LIN {X 0,Y 330.91,Z 992.639,A -85,B 0,C 180,E1 15009.118,E2 15009.118} C_VEL
LIN {X 0,Y 333.093,Z 983.84,A -85,B 0,C 180,E1 15005.534,E2 15005.534} C_VEL
LIN {X 0,Y 336.451,Z 972.211,A -85,B 0,C 180,E1 15001.598,E2 15001.598} C_VEL
LIN {X 0,Y 340.194,Z 960.433,A -85,B 0,C 180,E1 14998.264,E2 14998.264} C_VEL
LIN {X 0,Y 344.804,Z 946.621,A -85,B 0,C 180,E1 14994.966,E2 14994.966} C_VEL
LIN {X 0,Y 350.006,Z 931.551,A -85,B 0,C 180,E1 14991.906,E2 14991.906} C_VEL
LIN {X 0,Y 355.638,Z 914.95,A -85,B 0,C 180,E1 14989.083,E2 14989.083} C_VEL
LIN {X 0,Y 361.606,Z 897.07,A -85,B 0,C 180,E1 14986.496,E2 14986.496} C_VEL
LIN {X 0,Y 367.141,Z 879.555,A -85,B 0,C 180,E1 14984.374,E2 14984.374} C_VEL
LIN {X 0,Y 373.38,Z 858.51,A -85,B 0,C 180,E1 14982.232,E2 14982.232} C_VEL
LIN {X 0,Y 378.589,Z 839.318,A -85,B 0,C 180,E1 14980.607,E2 14980.607} C_VEL
LIN {X 0,Y 383.892,Z 817.228,A -85,B 0,C 180,E1 14979.071,E2 14979.071} C_VEL
LIN {X 0,Y 388.44,Z 795.784,A -85,B 0,C 180,E1 14977.862,E2 14977.862} C_VEL
LIN {X 0,Y 392.348,Z 773.028,A -85,B 0,C 180,E1 14976.87,E2 14976.87} C_VEL
LIN {X 0,Y 395.641,Z 749.252,A -85,B 0,C 180,E1 14976.094,E2 14976.094} C_VEL
LIN {X 0,Y 397.692,Z 726.736,A -85,B 0,C 180,E1 14975.556,E2 14975.556} C_VEL
LIN {X 0,Y 410.028,Z 517.167,A -85,B 0,C 180,E1 14971.398,E2 14971.398} C_VEL
LIN {X 0,Y 411.387,Z 493.975,A -85,B 0,C 180,E1 14970.919,E2 14970.919} C_VEL
LIN {X 0,Y 401.273,Z 477.851,A -85,B 0,C 180,E1 14968.094,E2 14968.094} C_VEL
LIN {X 0,Y 391.227,Z 463.001,A -85,B 0,C 180,E1 14964.981,E2 14964.981} C_VEL
LIN {X 0,Y 382.41,Z 450.658,A -85,B 0,C 180,E1 14961.915,E2 14961.915} C_VEL
LIN {X 0,Y 378.241,Z 445.412,A -85,B 0,C 180,E1 14960.341,E2 14960.341} C_VEL
LIN {X 0,Y 374.323,Z 440.519,A -85,B 0,C 180,E1 14958.775,E2 14958.775} C_VEL
LIN {X 0,Y 370.45,Z 435.602,A -85,B 0,C 180,E1 14957.109,E2 14957.109} C_VEL
LIN {X 0,Y 366.394,Z 431.101,A -85,B 0,C 180,E1 14955.268,E2 14955.268} C_VEL
LIN {X 0,Y 364.882,Z 429.094,A -85,B 0,C 180,E1 14954.52,E2 14954.52} C_VEL
LIN {X 0,Y 361.373,Z 425.41,A -85,B 0,C 180,E1 14952.747,E2 14952.747} C_VEL
LIN {X 0,Y 359.797,Z 423.107,A -85,B 0,C 180,E1 14951.867,E2 14951.867} C_VEL
LIN {X 0,Y 356.404,Z 419.891,A -85,B 0,C 180,E1 14949.935,E2 14949.935} C_VEL
LIN {X 0,Y 354.609,Z 416.906,A -85,B 0,C 180,E1 14948.757,E2 14948.757} C_VEL
LIN {X 0,Y 351.319,Z 414.41,A -85,B 0,C 180,E1 14946.618,E2 14946.618} C_VEL
LIN {X 0,Y 349.107,Z 410.908,A -85,B 0,C 180,E1 14944.887,E2 14944.887} C_VEL
LIN {X 0,Y 348.552,Z 410.26,A -85,B 0,C 180,E1 14944.442,E2 14944.442} C_VEL
LIN {X 0,Y 345.174,Z 407.913,A -85,B 0,C 180,E1 14941.659,E2 14941.659} C_VEL
LIN {X 0,Y 342.781,Z 403.846,A -85,B 0,C 180,E1 14938.997,E2 14938.997} C_VEL
LIN {X 0,Y 338.729,Z 401.153,A -85,B 0,C 180,E1 14933.729,E2 14933.729} C_VEL
LIN {X 0,Y 336.722,Z 397.551,A -85,B 0,C 180,E1 14928.46,E2 14928.46} C_VEL
LIN {X 0,Y 336.018,Z 396.934,A -85,B 0,C 180,E1 14923.757,E2 14923.757} C_VEL
LIN {X 0,Y 336.593,Z 397.417,A -85,B 0,C 180,E1 14919.116,E2 14919.116} C_VEL
LIN {X 0,Y 337.44,Z 399.091,A -85,B 0,C 180,E1 14916.235,E2 14916.235} C_VEL
LIN {X 0,Y 340.379,Z 402.576,A -85,B 0,C 180,E1 14911.008,E2 14911.008} C_VEL
LIN {X 0,Y 343.088,Z 404.15,A -85,B 0,C 180,E1 14907.868,E2 14907.868} C_VEL
LIN {X 0,Y 345.313,Z 408.031,A -85,B 0,C 180,E1 14905.422,E2 14905.422} C_VEL
LIN {X 0,Y 349.089,Z 410.785,A -85,B 0,C 180,E1 14902.353,E2 14902.353} C_VEL
LIN {X 0,Y 351.324,Z 414.39,A -85,B 0,C 180,E1 14900.605,E2 14900.605} C_VEL
LIN {X 0,Y 354.877,Z 417.344,A -85,B 0,C 180,E1 14898.291,E2 14898.291} C_VEL
LIN {X 0,Y 357.657,Z 421.353,A -85,B 0,C 180,E1 14896.55,E2 14896.55} C_VEL
LIN {X 0,Y 360.381,Z 423.715,A -85,B 0,C 180,E1 14895.07,E2 14895.07} C_VEL
LIN {X 0,Y 363.451,Z 427.853,A -85,B 0,C 180,E1 14893.425,E2 14893.425} C_VEL
LIN {X 0,Y 365.762,Z 430.068,A -85,B 0,C 180,E1 14892.315,E2 14892.315} C_VEL
LIN {X 0,Y 369.415,Z 434.618,A -85,B 0,C 180,E1 14890.606,E2 14890.606} C_VEL
LIN {X 0,Y 371.075,Z 436.552,A -85,B 0,C 180,E1 14889.881,E2 14889.881} C_VEL
LIN {X 0,Y 375.981,Z 442.563,A -85,B 0,C 180,E1 14887.83,E2 14887.83} C_VEL
LIN {X 0,Y 380.704,Z 448.431,A -85,B 0,C 180,E1 14886.009,E2 14886.009} C_VEL
LIN {X 0,Y 385.386,Z 454.312,A -85,B 0,C 180,E1 14884.335,E2 14884.335} C_VEL
LIN {X 0,Y 393.083,Z 464.398,A -85,B 0,C 180,E1 14881.786,E2 14881.786} C_VEL
LIN {X 0,Y 402.393,Z 477.147,A -85,B 0,C 180,E1 14878.996,E2 14878.996} C_VEL
LIN {X 0,Y 411.104,Z 489.93,A -85,B 0,C 180,E1 14876.615,E2 14876.615} C_VEL
LIN {X 0,Y 398.81,Z 697.255,A -85,B 0,C 180,E1 14872.515,E2 14872.515} C_VEL
LIN {X 0,Y 396.721,Z 724.489,A -85,B 0,C 180,E1 14871.906,E2 14871.906} C_VEL
LIN {X 0,Y 393.982,Z 747.489,A -85,B 0,C 180,E1 14871.191,E2 14871.191} C_VEL
LIN {X 0,Y 390.444,Z 769.449,A -85,B 0,C 180,E1 14870.259,E2 14870.259} C_VEL
LIN {X 0,Y 386.299,Z 791.019,A -85,B 0,C 180,E1 14869.107,E2 14869.107} C_VEL
LIN {X 0,Y 381.676,Z 811.199,A -85,B 0,C 180,E1 14867.765,E2 14867.765} C_VEL
LIN {X 0,Y 376.156,Z 832.56,A -85,B 0,C 180,E1 14866.043,E2 14866.043} C_VEL
LIN {X 0,Y 370.908,Z 850.781,A -85,B 0,C 180,E1 14864.275,E2 14864.275} C_VEL
LIN {X 0,Y 364.791,Z 870.313,A -85,B 0,C 180,E1 14862.019,E2 14862.019} C_VEL
LIN {X 0,Y 359.17,Z 887.26,A -85,B 0,C 180,E1 14859.691,E2 14859.691} C_VEL
LIN {X 0,Y 355.793,Z 896.961,A -85,B 0,C 180,E1 14858.165,E2 14858.165} C_VEL
LIN {X 0,Y 353.148,Z 902.367,A -85,B 0,C 180,E1 14857.37,E2 14857.37} C_VEL
LIN {X 0,Y 343.413,Z 915.776,A -85,B 0,C 180,E1 14855.488,E2 14855.488} C_VEL
LIN {X 0,Y 340.743,Z 920.57,A -85,B 0,C 180,E1 14854.568,E2 14854.568} C_VEL
LIN {X 0,Y 335.906,Z 933.491,A -85,B 0,C 180,E1 14851.531,E2 14851.531} C_VEL
LIN {X 0,Y 330.984,Z 947.025,A -85,B 0,C 180,E1 14847.745,E2 14847.745} C_VEL
LIN {X 0,Y 327.238,Z 958.049,A -85,B 0,C 180,E1 14844.033,E2 14844.033} C_VEL
LIN {X 0,Y 324.369,Z 967.228,A -85,B 0,C 180,E1 14840.235,E2 14840.235} C_VEL
LIN {X 0,Y 322.352,Z 974.985,A -85,B 0,C 180,E1 14836.361,E2 14836.361} C_VEL
LIN {X 0,Y 321.026,Z 981.137,A -85,B 0,C 180,E1 14832.376,E2 14832.376} C_VEL
LIN {X 0,Y 320.326,Z 985.864,A -85,B 0,C 180,E1 14828.384,E2 14828.384} C_VEL
LIN {X 0,Y 320.045,Z 988.794,A -85,B 0,C 180,E1 14824.655,E2 14824.655} C_VEL
LIN {X 0,Y 319.986,Z 990.509,A -85,B 0,C 180,E1 14821.027,E2 14821.027} C_VEL
LIN {X 0,Y 319.956,Z 990.924,A -85,B 0,C 180,E1 14817.057,E2 14817.057} C_VEL
LIN {X 0,Y 319.974,Z 990.17,A -85,B 0,C 180,E1 14813.727,E2 14813.727} C_VEL
LIN {X 0,Y 320.14,Z 988.143,A -85,B 0,C 180,E1 14809.924,E2 14809.924} C_VEL
LIN {X 0,Y 320.531,Z 984.612,A -85,B 0,C 180,E1 14806.103,E2 14806.103} C_VEL
LIN {X 0,Y 321.437,Z 979.74,A -85,B 0,C 180,E1 14802.214,E2 14802.214} C_VEL
LIN {X 0,Y 322.994,Z 973.105,A -85,B 0,C 180,E1 14798.253,E2 14798.253} C_VEL
LIN {X 0,Y 325.442,Z 964.846,A -85,B 0,C 180,E1 14794.259,E2 14794.259} C_VEL
LIN {X 0,Y 328.74,Z 954.945,A -85,B 0,C 180,E1 14790.426,E2 14790.426} C_VEL
LIN {X 0,Y 333.353,Z 942.442,A -85,B 0,C 180,E1 14786.423,E2 14786.423} C_VEL
LIN {X 0,Y 338.143,Z 930.095,A -85,B 0,C 180,E1 14783.126,E2 14783.126} C_VEL
LIN {X 0,Y 343.659,Z 916.024,A -85,B 0,C 180,E1 14779.983,E2 14779.983} C_VEL
LIN {X 0,Y 349.738,Z 900.54,A -85,B 0,C 180,E1 14777.04,E2 14777.04} C_VEL
LIN {X 0,Y 355.801,Z 884.413,A -85,B 0,C 180,E1 14774.484,E2 14774.484} C_VEL
LIN {X 0,Y 362.443,Z 866.085,A -85,B 0,C 180,E1 14772.022,E2 14772.022} C_VEL
LIN {X 0,Y 368.203,Z 848.908,A -85,B 0,C 180,E1 14770.088,E2 14770.088} C_VEL
LIN {X 0,Y 374.697,Z 827.854,A -85,B 0,C 180,E1 14768.099,E2 14768.099} C_VEL
LIN {X 0,Y 380.15,Z 808.098,A -85,B 0,C 180,E1 14766.563,E2 14766.563} C_VEL
LIN {X 0,Y 385.245,Z 786.857,A -85,B 0,C 180,E1 14765.212,E2 14765.212} C_VEL
LIN {X 0,Y 389.81,Z 764.653,A -85,B 0,C 180,E1 14764.078,E2 14764.078} C_VEL
LIN {X 0,Y 393.502,Z 741.577,A -85,B 0,C 180,E1 14763.184,E2 14763.184} C_VEL
LIN {X 0,Y 396.477,Z 716.689,A -85,B 0,C 180,E1 14762.486,E2 14762.486} C_VEL
LIN {X 0,Y 412.263,Z 510.138,A -85,B 0,C 180,E1 14758.198,E2 14758.198} C_VEL
LIN {X 0,Y 413.31,Z 496.471,A -85,B 0,C 180,E1 14757.89,E2 14757.89} C_VEL
LIN {X 0,Y 407.813,Z 487.013,A -85,B 0,C 180,E1 14755.501,E2 14755.501} C_VEL
LIN {X 0,Y 403.867,Z 480.436,A -85,B 0,C 180,E1 14753.39,E2 14753.39} C_VEL
LIN {X 0,Y 401.279,Z 476.234,A -85,B 0,C 180,E1 14751.691,E2 14751.691} C_VEL
LIN {X 0,Y 398.884,Z 472.1,A -85,B 0,C 180,E1 14749.603,E2 14749.603} C_VEL
LIN {X 0,Y 396.705,Z 468.572,A -85,B 0,C 180,E1 14746.444,E2 14746.444} C_VEL
LIN {X 0,Y 396.482,Z 467.384,A -85,B 0,C 180,E1 14745.394,E2 14745.394} C_VEL
LIN {X 0,Y 396.528,Z 467.443,A -85,B 0,C 180,E1 14742.842,E2 14742.842} C_VEL
LIN {X 0,Y 398.037,Z 471.243,A -85,B 0,C 180,E1 14739.718,E2 14739.718} C_VEL
LIN {X 0,Y 399.24,Z 472.726,A -85,B 0,C 180,E1 14738.476,E2 14738.476} C_VEL
LIN {X 0,Y 402.217,Z 477.734,A -85,B 0,C 180,E1 14736.097,E2 14736.097} C_VEL
LIN {X 0,Y 405.36,Z 483.575,A -85,B 0,C 180,E1 14734.157,E2 14734.157} C_VEL
LIN {X 0,Y 409.464,Z 491.64,A -85,B 0,C 180,E1 14732.085,E2 14732.085} C_VEL
LIN {X 0,Y 413.288,Z 499.593,A -85,B 0,C 180,E1 14730.423,E2 14730.423} C_VEL
LIN {X 0,Y 399.434,Z 680.245,A -85,B 0,C 180,E1 14726.677,E2 14726.677} C_VEL
LIN {X 0,Y 395.3,Z 735.513,A -85,B 0,C 180,E1 14725.506,E2 14725.506} C_VEL
LIN {X 0,Y 392.181,Z 758.741,A -85,B 0,C 180,E1 14724.843,E2 14724.843} C_VEL
LIN {X 0,Y 388.044,Z 782.281,A -85,B 0,C 180,E1 14723.946,E2 14723.946} C_VEL
LIN {X 0,Y 383.894,Z 801.848,A -85,B 0,C 180,E1 14722.983,E2 14722.983} C_VEL
LIN {X 0,Y 378.352,Z 824.459,A -85,B 0,C 180,E1 14721.591,E2 14721.591} C_VEL
LIN {X 0,Y 373.178,Z 843.178,A -85,B 0,C 180,E1 14720.182,E2 14720.182} C_VEL
LIN {X 0,Y 366.642,Z 864.591,A -85,B 0,C 180,E1 14718.236,E2 14718.236} C_VEL
LIN {X 0,Y 360.423,Z 883.572,A -85,B 0,C 180,E1 14716.164,E2 14716.164} C_VEL
LIN {X 0,Y 354.049,Z 901.749,A -85,B 0,C 180,E1 14713.784,E2 14713.784} C_VEL
LIN {X 0,Y 347.941,Z 918.842,A -85,B 0,C 180,E1 14711.156,E2 14711.156} C_VEL
LIN {X 0,Y 341.813,Z 935.354,A -85,B 0,C 180,E1 14708.117,E2 14708.117} C_VEL
LIN {X 0,Y 336.304,Z 950.548,A -85,B 0,C 180,E1 14704.812,E2 14704.812} C_VEL
LIN {X 0,Y 331.687,Z 963.637,A -85,B 0,C 180,E1 14701.437,E2 14701.437} C_VEL
LIN {X 0,Y 327.626,Z 975.984,A -85,B 0,C 180,E1 14697.642,E2 14697.642} C_VEL
LIN {X 0,Y 324.704,Z 985.988,A -85,B 0,C 180,E1 14693.987,E2 14693.987} C_VEL
LIN {X 0,Y 322.437,Z 995.015,A -85,B 0,C 180,E1 14689.948,E2 14689.948} C_VEL
LIN {X 0,Y 321.025,Z 1002.362,A -85,B 0,C 180,E1 14685.912,E2 14685.912} C_VEL
LIN {X 0,Y 320.293,Z 1007.625,A -85,B 0,C 180,E1 14682.077,E2 14682.077} C_VEL
LIN {X 0,Y 320.032,Z 1011.372,A -85,B 0,C 180,E1 14678.448,E2 14678.448} C_VEL
LIN {X 0,Y 319.948,Z 1013.912,A -85,B 0,C 180,E1 14674.485,E2 14674.485} C_VEL
LIN {X 0,Y 319.955,Z 1014.848,A -85,B 0,C 180,E1 14671.258,E2 14671.258} C_VEL
LIN {X 0,Y 319.957,Z 1014.757,A -85,B 0,C 180,E1 14667.856,E2 14667.856} C_VEL
LIN {X 0,Y 319.959,Z 1013.149,A -85,B 0,C 180,E1 14663.906,E2 14663.906} C_VEL
LIN {X 0,Y 320.069,Z 1010.511,A -85,B 0,C 180,E1 14660.475,E2 14660.475} C_VEL
LIN {X 0,Y 320.522,Z 1006.032,A -85,B 0,C 180,E1 14656.475,E2 14656.475} C_VEL
LIN {X 0,Y 321.456,Z 1000.106,A -85,B 0,C 180,E1 14652.632,E2 14652.632} C_VEL
LIN {X 0,Y 323.158,Z 992.282,A -85,B 0,C 180,E1 14648.592,E2 14648.592} C_VEL
LIN {X 0,Y 325.502,Z 983.467,A -85,B 0,C 180,E1 14644.925,E2 14644.925} C_VEL
LIN {X 0,Y 329.077,Z 971.865,A -85,B 0,C 180,E1 14640.919,E2 14640.919} C_VEL
LIN {X 0,Y 333.072,Z 960.003,A -85,B 0,C 180,E1 14637.504,E2 14637.504} C_VEL
LIN {X 0,Y 337.94,Z 946.141,A -85,B 0,C 180,E1 14634.146,E2 14634.146} C_VEL
LIN {X 0,Y 343.504,Z 930.845,A -85,B 0,C 180,E1 14631.002,E2 14631.002} C_VEL
LIN {X 0,Y 349.325,Z 914.383,A -85,B 0,C 180,E1 14628.179,E2 14628.179} C_VEL
LIN {X 0,Y 355.575,Z 896.402,A -85,B 0,C 180,E1 14625.567,E2 14625.567} C_VEL
LIN {X 0,Y 361.579,Z 878.166,A -85,B 0,C 180,E1 14623.351,E2 14623.351} C_VEL
LIN {X 0,Y 367.893,Z 857.519,A -85,B 0,C 180,E1 14621.254,E2 14621.254} C_VEL
LIN {X 0,Y 373.243,Z 838.445,A -85,B 0,C 180,E1 14619.64,E2 14619.64} C_VEL
LIN {X 0,Y 378.399,Z 817.624,A -85,B 0,C 180,E1 14618.192,E2 14618.192} C_VEL
LIN {X 0,Y 383.162,Z 795.876,A -85,B 0,C 180,E1 14616.96,E2 14616.96} C_VEL
LIN {X 0,Y 387.235,Z 772.987,A -85,B 0,C 180,E1 14615.957,E2 14615.957} C_VEL
LIN {X 0,Y 390.634,Z 749.321,A -85,B 0,C 180,E1 14615.182,E2 14615.182} C_VEL
LIN {X 0,Y 392.766,Z 726.741,A -85,B 0,C 180,E1 14614.638,E2 14614.638} C_VEL
LIN {X 0,Y 405.62,Z 516.743,A -85,B 0,C 180,E1 14610.449,E2 14610.449} C_VEL
LIN {X 0,Y 406.726,Z 498.175,A -85,B 0,C 180,E1 14610.062,E2 14610.062} C_VEL
LIN {X 0,Y 397.976,Z 484.066,A -85,B 0,C 180,E1 14607.533,E2 14607.533} C_VEL
LIN {X 0,Y 388.403,Z 469.686,A -85,B 0,C 180,E1 14604.485,E2 14604.485} C_VEL
LIN {X 0,Y 379.904,Z 457.646,A -85,B 0,C 180,E1 14601.458,E2 14601.458} C_VEL
LIN {X 0,Y 375.865,Z 452.522,A -85,B 0,C 180,E1 14599.907,E2 14599.907} C_VEL
LIN {X 0,Y 372.014,Z 447.669,A -85,B 0,C 180,E1 14598.328,E2 14598.328} C_VEL
LIN {X 0,Y 367.517,Z 442.164,A -85,B 0,C 180,E1 14596.354,E2 14596.354} C_VEL
LIN {X 0,Y 363.777,Z 437.473,A -85,B 0,C 180,E1 14594.565,E2 14594.565} C_VEL
LIN {X 0,Y 359.268,Z 432.497,A -85,B 0,C 180,E1 14592.251,E2 14592.251} C_VEL
LIN {X 0,Y 358.132,Z 430.776,A -85,B 0,C 180,E1 14591.596,E2 14591.596} C_VEL
LIN {X 0,Y 354.635,Z 427.367,A -85,B 0,C 180,E1 14589.575,E2 14589.575} C_VEL
LIN {X 0,Y 352.73,Z 424.487,A -85,B 0,C 180,E1 14588.312,E2 14588.312} C_VEL
LIN {X 0,Y 349.419,Z 421.648,A -85,B 0,C 180,E1 14586.077,E2 14586.077} C_VEL
LIN {X 0,Y 347.235,Z 418.11,A -85,B 0,C 180,E1 14584.293,E2 14584.293} C_VEL
LIN {X 0,Y 343.702,Z 415.553,A -85,B 0,C 180,E1 14581.333,E2 14581.333} C_VEL
LIN {X 0,Y 341.496,Z 411.677,A -85,B 0,C 180,E1 14578.825,E2 14578.825} C_VEL
LIN {X 0,Y 337.513,Z 408.987,A -85,B 0,C 180,E1 14573.536,E2 14573.536} C_VEL
LIN {X 0,Y 335.565,Z 405.439,A -85,B 0,C 180,E1 14568.31,E2 14568.31} C_VEL
LIN {X 0,Y 334.91,Z 404.851,A -85,B 0,C 180,E1 14563.523,E2 14563.523} C_VEL
LIN {X 0,Y 335.611,Z 405.454,A -85,B 0,C 180,E1 14558.686,E2 14558.686} C_VEL
LIN {X 0,Y 338.405,Z 409.854,A -85,B 0,C 180,E1 14552.171,E2 14552.171} C_VEL
LIN {X 0,Y 341.724,Z 411.891,A -85,B 0,C 180,E1 14548.12,E2 14548.12} C_VEL
LIN {X 0,Y 343.957,Z 415.81,A -85,B 0,C 180,E1 14545.635,E2 14545.635} C_VEL
LIN {X 0,Y 347.537,Z 418.459,A -85,B 0,C 180,E1 14542.675,E2 14542.675} C_VEL
LIN {X 0,Y 350.003,Z 422.307,A -85,B 0,C 180,E1 14540.72,E2 14540.72} C_VEL
LIN {X 0,Y 353.228,Z 425.038,A -85,B 0,C 180,E1 14538.592,E2 14538.592} C_VEL
LIN {X 0,Y 356.131,Z 429.107,A -85,B 0,C 180,E1 14536.76,E2 14536.76} C_VEL
LIN {X 0,Y 358.645,Z 431.399,A -85,B 0,C 180,E1 14535.368,E2 14535.368} C_VEL
LIN {X 0,Y 361.874,Z 435.618,A -85,B 0,C 180,E1 14533.621,E2 14533.621} C_VEL
LIN {X 0,Y 363.902,Z 437.65,A -85,B 0,C 180,E1 14532.635,E2 14532.635} C_VEL
LIN {X 0,Y 367.605,Z 442.217,A -85,B 0,C 180,E1 14530.874,E2 14530.874} C_VEL
LIN {X 0,Y 373.794,Z 449.865,A -85,B 0,C 180,E1 14528.209,E2 14528.209} C_VEL
LIN {X 0,Y 378.705,Z 456.06,A -85,B 0,C 180,E1 14526.286,E2 14526.286} C_VEL
LIN {X 0,Y 383.771,Z 462.499,A -85,B 0,C 180,E1 14524.452,E2 14524.452} C_VEL
LIN {X 0,Y 393.127,Z 474.956,A -85,B 0,C 180,E1 14521.358,E2 14521.358} C_VEL
LIN {X 0,Y 403.739,Z 490.155,A -85,B 0,C 180,E1 14518.225,E2 14518.225} C_VEL
LIN {X 0,Y 406.441,Z 494.536,A -85,B 0,C 180,E1 14517.468,E2 14517.468} C_VEL
LIN {X 0,Y 393.64,Z 702.589,A -85,B 0,C 180,E1 14513.331,E2 14513.331} C_VEL
LIN {X 0,Y 391.59,Z 726.521,A -85,B 0,C 180,E1 14512.772,E2 14512.772} C_VEL
LIN {X 0,Y 388.641,Z 749.694,A -85,B 0,C 180,E1 14512.027,E2 14512.027} C_VEL
LIN {X 0,Y 385.198,Z 770.255,A -85,B 0,C 180,E1 14511.144,E2 14511.144} C_VEL
LIN {X 0,Y 380.794,Z 792.284,A -85,B 0,C 180,E1 14509.954,E2 14509.954} C_VEL
LIN {X 0,Y 376.03,Z 812.406,A -85,B 0,C 180,E1 14508.602,E2 14508.602} C_VEL
LIN {X 0,Y 370.317,Z 833.635,A -85,B 0,C 180,E1 14506.868,E2 14506.868} C_VEL
LIN {X 0,Y 364.887,Z 851.797,A -85,B 0,C 180,E1 14505.084,E2 14505.084} C_VEL
LIN {X 0,Y 358.535,Z 871.225,A -85,B 0,C 180,E1 14502.804,E2 14502.804} C_VEL
LIN {X 0,Y 352.523,Z 888.687,A -85,B 0,C 180,E1 14500.371,E2 14500.371} C_VEL
LIN {X 0,Y 346.505,Z 905.102,A -85,B 0,C 180,E1 14497.623,E2 14497.623} C_VEL
LIN {X 0,Y 340.743,Z 920.57,A -85,B 0,C 180,E1 14494.568,E2 14494.568} C_VEL
LIN {X 0,Y 338.108,Z 925.306,A -85,B 0,C 180,E1 14493.617,E2 14493.617} C_VEL
LIN {X 0,Y 328.091,Z 937.671,A -85,B 0,C 180,E1 14491.193,E2 14491.193} C_VEL
LIN {X 0,Y 326.075,Z 941.156,A -85,B 0,C 180,E1 14490.277,E2 14490.277} C_VEL
LIN {X 0,Y 321.565,Z 953.258,A -85,B 0,C 180,E1 14486.478,E2 14486.478} C_VEL
LIN {X 0,Y 318.181,Z 962.982,A -85,B 0,C 180,E1 14482.775,E2 14482.775} C_VEL
LIN {X 0,Y 315.454,Z 971.82,A -85,B 0,C 180,E1 14478.662,E2 14478.662} C_VEL
LIN {X 0,Y 313.768,Z 978.407,A -85,B 0,C 180,E1 14474.848,E2 14474.848} C_VEL
LIN {X 0,Y 312.666,Z 984.079,A -85,B 0,C 180,E1 14470.57,E2 14470.57} C_VEL
LIN {X 0,Y 312.184,Z 987.545,A -85,B 0,C 180,E1 14466.995,E2 14466.995} C_VEL
LIN {X 0,Y 311.992,Z 990.13,A -85,B 0,C 180,E1 14462.926,E2 14462.926} C_VEL
LIN {X 0,Y 311.962,Z 991.137,A -85,B 0,C 180,E1 14459.358,E2 14459.358} C_VEL
LIN {X 0,Y 311.954,Z 991.102,A -85,B 0,C 180,E1 14455.877,E2 14455.877} C_VEL
LIN {X 0,Y 312.03,Z 989.685,A -85,B 0,C 180,E1 14451.793,E2 14451.793} C_VEL
LIN {X 0,Y 312.28,Z 987.245,A -85,B 0,C 180,E1 14448.238,E2 14448.238} C_VEL
LIN {X 0,Y 312.926,Z 983.148,A -85,B 0,C 180,E1 14444.152,E2 14444.152} C_VEL
LIN {X 0,Y 314.157,Z 977.592,A -85,B 0,C 180,E1 14440.191,E2 14440.191} C_VEL
LIN {X 0,Y 316.149,Z 970.673,A -85,B 0,C 180,E1 14436.243,E2 14436.243} C_VEL
LIN {X 0,Y 319.124,Z 961.659,A -85,B 0,C 180,E1 14432.184,E2 14432.184} C_VEL
LIN {X 0,Y 323.341,Z 950.407,A -85,B 0,C 180,E1 14428.037,E2 14428.037} C_VEL
LIN {X 0,Y 328.198,Z 938.354,A -85,B 0,C 180,E1 14424.363,E2 14424.363} C_VEL
LIN {X 0,Y 333.708,Z 924.882,A -85,B 0,C 180,E1 14420.97,E2 14420.97} C_VEL
LIN {X 0,Y 339.902,Z 910.055,A -85,B 0,C 180,E1 14417.815,E2 14417.815} C_VEL
LIN {X 0,Y 346.137,Z 894.608,A -85,B 0,C 180,E1 14415.069,E2 14415.069} C_VEL
LIN {X 0,Y 353.157,Z 876.566,A -85,B 0,C 180,E1 14412.365,E2 14412.365} C_VEL
LIN {X 0,Y 359.885,Z 858.283,A -85,B 0,C 180,E1 14410.081,E2 14410.081} C_VEL
LIN {X 0,Y 366.401,Z 838.867,A -85,B 0,C 180,E1 14408.071,E2 14408.071} C_VEL
LIN {X 0,Y 372.65,Z 818.56,A -85,B 0,C 180,E1 14406.316,E2 14406.316} C_VEL
LIN {X 0,Y 377.881,Z 798.972,A -85,B 0,C 180,E1 14404.934,E2 14404.934} C_VEL
LIN {X 0,Y 382.988,Z 777.255,A -85,B 0,C 180,E1 14403.675,E2 14403.675} C_VEL
LIN {X 0,Y 386.924,Z 756.792,A -85,B 0,C 180,E1 14402.741,E2 14402.741} C_VEL
LIN {X 0,Y 390.481,Z 733.779,A -85,B 0,C 180,E1 14401.93,E2 14401.93} C_VEL
LIN {X 0,Y 392.861,Z 711.932,A -85,B 0,C 180,E1 14401.37,E2 14401.37} C_VEL
LIN {X 0,Y 408.594,Z 515.485,A -85,B 0,C 180,E1 14397.28,E2 14397.28} C_VEL
LIN {X 0,Y 409.73,Z 501.348,A -85,B 0,C 180,E1 14396.958,E2 14396.958} C_VEL
LIN {X 0,Y 404.903,Z 492.579,A -85,B 0,C 180,E1 14394.652,E2 14394.652} C_VEL
LIN {X 0,Y 401.655,Z 487.205,A -85,B 0,C 180,E1 14392.779,E2 14392.779} C_VEL
LIN {X 0,Y 399.671,Z 483.764,A -85,B 0,C 180,E1 14391.368,E2 14391.368} C_VEL
LIN {X 0,Y 397.398,Z 479.759,A -85,B 0,C 180,E1 14389.27,E2 14389.27} C_VEL
LIN {X 0,Y 395.488,Z 476.165,A -85,B 0,C 180,E1 14386.104,E2 14386.104} C_VEL
LIN {X 0,Y 395.315,Z 475.274,A -85,B 0,C 180,E1 14385.2,E2 14385.2} C_VEL
LIN {X 0,Y 395.397,Z 475.527,A -85,B 0,C 180,E1 14382.791,E2 14382.791} C_VEL
LIN {X 0,Y 396.825,Z 479.135,A -85,B 0,C 180,E1 14379.807,E2 14379.807} C_VEL
LIN {X 0,Y 397.842,Z 480.472,A -85,B 0,C 180,E1 14378.706,E2 14378.706} C_VEL
LIN {X 0,Y 400.591,Z 485.328,A -85,B 0,C 180,E1 14376.385,E2 14376.385} C_VEL
LIN {X 0,Y 403.576,Z 491.165,A -85,B 0,C 180,E1 14374.464,E2 14374.464} C_VEL
LIN {X 0,Y 407.452,Z 499.153,A -85,B 0,C 180,E1 14372.408,E2 14372.408} C_VEL
LIN {X 0,Y 409.694,Z 504.249,A -85,B 0,C 180,E1 14371.353,E2 14371.353} C_VEL
LIN {X 0,Y 395.083,Z 685.929,A -85,B 0,C 180,E1 14367.569,E2 14367.569} C_VEL
LIN {X 0,Y 391.175,Z 735.184,A -85,B 0,C 180,E1 14366.514,E2 14366.514} C_VEL
LIN {X 0,Y 387.901,Z 758.589,A -85,B 0,C 180,E1 14365.846,E2 14365.846} C_VEL
LIN {X 0,Y 383.73,Z 781.545,A -85,B 0,C 180,E1 14364.977,E2 14364.977} C_VEL
LIN {X 0,Y 379.343,Z 801.417,A -85,B 0,C 180,E1 14364.001,E2 14364.001} C_VEL
LIN {X 0,Y 373.419,Z 824.628,A -85,B 0,C 180,E1 14362.569,E2 14362.569} C_VEL
LIN {X 0,Y 368.206,Z 842.703,A -85,B 0,C 180,E1 14361.204,E2 14361.204} C_VEL
LIN {X 0,Y 361.315,Z 864.379,A -85,B 0,C 180,E1 14359.227,E2 14359.227} C_VEL
LIN {X 0,Y 355.226,Z 882.134,A -85,B 0,C 180,E1 14357.281,E2 14357.281} C_VEL
LIN {X 0,Y 348.46,Z 900.631,A -85,B 0,C 180,E1 14354.869,E2 14354.869} C_VEL
LIN {X 0,Y 342.073,Z 917.596,A -85,B 0,C 180,E1 14352.247,E2 14352.247} C_VEL
LIN {X 0,Y 335.789,Z 933.754,A -85,B 0,C 180,E1 14349.27,E2 14349.27} C_VEL
LIN {X 0,Y 330.01,Z 948.825,A -85,B 0,C 180,E1 14346.004,E2 14346.004} C_VEL
LIN {X 0,Y 324.975,Z 962.151,A -85,B 0,C 180,E1 14342.541,E2 14342.541} C_VEL
LIN {X 0,Y 320.412,Z 975.142,A -85,B 0,C 180,E1 14338.523,E2 14338.523} C_VEL
LIN {X 0,Y 317.232,Z 985.195,A -85,B 0,C 180,E1 14334.788,E2 14334.788} C_VEL
LIN {X 0,Y 314.748,Z 994.332,A -85,B 0,C 180,E1 14330.652,E2 14330.652} C_VEL
LIN {X 0,Y 313.24,Z 1001.428,A -85,B 0,C 180,E1 14326.699,E2 14326.699} C_VEL
LIN {X 0,Y 312.365,Z 1007.098,A -85,B 0,C 180,E1 14322.576,E2 14322.576} C_VEL
LIN {X 0,Y 312.044,Z 1010.899,A -85,B 0,C 180,E1 14318.852,E2 14318.852} C_VEL
LIN {X 0,Y 311.951,Z 1013.537,A -85,B 0,C 180,E1 14314.785,E2 14314.785} C_VEL
LIN {X 0,Y 311.961,Z 1014.548,A -85,B 0,C 180,E1 14311.29,E2 14311.29} C_VEL
LIN {X 0,Y 311.961,Z 1014.457,A -85,B 0,C 180,E1 14307.801,E2 14307.801} C_VEL
LIN {X 0,Y 311.96,Z 1012.96,A -85,B 0,C 180,E1 14303.934,E2 14303.934} C_VEL
LIN {X 0,Y 312.071,Z 1010.365,A -85,B 0,C 180,E1 14300.415,E2 14300.415} C_VEL
LIN {X 0,Y 312.514,Z 1006.211,A -85,B 0,C 180,E1 14296.499,E2 14296.499} C_VEL
LIN {X 0,Y 313.496,Z 1000.261,A -85,B 0,C 180,E1 14292.48,E2 14292.48} C_VEL
LIN {X 0,Y 315.232,Z 992.754,A -85,B 0,C 180,E1 14288.418,E2 14288.418} C_VEL
LIN {X 0,Y 317.801,Z 983.563,A -85,B 0,C 180,E1 14284.474,E2 14284.474} C_VEL
LIN {X 0,Y 321.373,Z 972.624,A -85,B 0,C 180,E1 14280.563,E2 14280.563} C_VEL
LIN {X 0,Y 325.513,Z 960.868,A -85,B 0,C 180,E1 14277.072,E2 14277.072} C_VEL
LIN {X 0,Y 330.856,Z 946.452,A -85,B 0,C 180,E1 14273.47,E2 14273.47} C_VEL
LIN {X 0,Y 336.237,Z 932.256,A -85,B 0,C 180,E1 14270.486,E2 14270.486} C_VEL
LIN {X 0,Y 342.34,Z 915.864,A -85,B 0,C 180,E1 14267.579,E2 14267.579} C_VEL
LIN {X 0,Y 348.796,Z 898.22,A -85,B 0,C 180,E1 14264.932,E2 14264.932} C_VEL
LIN {X 0,Y 354.97,Z 880.181,A -85,B 0,C 180,E1 14262.687,E2 14262.687} C_VEL
LIN {X 0,Y 361.156,Z 861.057,A -85,B 0,C 180,E1 14260.671,E2 14260.671} C_VEL
LIN {X 0,Y 366.7,Z 842.087,A -85,B 0,C 180,E1 14259.014,E2 14259.014} C_VEL
LIN {X 0,Y 372.281,Z 821.059,A -85,B 0,C 180,E1 14257.482,E2 14257.482} C_VEL
LIN {X 0,Y 376.991,Z 800.512,A -85,B 0,C 180,E1 14256.276,E2 14256.276} C_VEL
LIN {X 0,Y 381.514,Z 777.268,A -85,B 0,C 180,E1 14255.191,E2 14255.191} C_VEL
LIN {X 0,Y 384.863,Z 755.951,A -85,B 0,C 180,E1 14254.44,E2 14254.44} C_VEL
LIN {X 0,Y 387.578,Z 731.322,A -85,B 0,C 180,E1 14253.8,E2 14253.8} C_VEL
LIN {X 0,Y 400.92,Z 522.223,A -85,B 0,C 180,E1 14249.599,E2 14249.599} C_VEL
LIN {X 0,Y 402.113,Z 502.251,A -85,B 0,C 180,E1 14249.166,E2 14249.166} C_VEL
LIN {X 0,Y 393.667,Z 488.63,A -85,B 0,C 180,E1 14246.633,E2 14246.633} C_VEL
LIN {X 0,Y 384.148,Z 474.161,A -85,B 0,C 180,E1 14243.467,E2 14243.467} C_VEL
LIN {X 0,Y 374.88,Z 461.116,A -85,B 0,C 180,E1 14240.002,E2 14240.002} C_VEL
LIN {X 0,Y 369.37,Z 454.437,A -85,B 0,C 180,E1 14237.729,E2 14237.729} C_VEL
LIN {X 0,Y 365.453,Z 449.507,A -85,B 0,C 180,E1 14235.959,E2 14235.959} C_VEL
LIN {X 0,Y 360.997,Z 444.014,A -85,B 0,C 180,E1 14233.779,E2 14233.779} C_VEL
LIN {X 0,Y 357.319,Z 439.789,A -85,B 0,C 180,E1 14231.827,E2 14231.827} C_VEL
LIN {X 0,Y 356.044,Z 438.141,A -85,B 0,C 180,E1 14231.09,E2 14231.09} C_VEL
LIN {X 0,Y 352.519,Z 434.318,A -85,B 0,C 180,E1 14228.974,E2 14228.974} C_VEL
LIN {X 0,Y 351.127,Z 432.191,A -85,B 0,C 180,E1 14228.02,E2 14228.02} C_VEL
LIN {X 0,Y 347.75,Z 429.143,A -85,B 0,C 180,E1 14225.692,E2 14225.692} C_VEL
LIN {X 0,Y 345.701,Z 425.858,A -85,B 0,C 180,E1 14223.98,E2 14223.98} C_VEL
LIN {X 0,Y 342.323,Z 423.295,A -85,B 0,C 180,E1 14221.087,E2 14221.087} C_VEL
LIN {X 0,Y 340.036,Z 419.396,A -85,B 0,C 180,E1 14218.461,E2 14218.461} C_VEL
LIN {X 0,Y 336.301,Z 416.82,A -85,B 0,C 180,E1 14213.341,E2 14213.341} C_VEL
LIN {X 0,Y 334.44,Z 413.356,A -85,B 0,C 180,E1 14208.27,E2 14208.27} C_VEL
LIN {X 0,Y 333.804,Z 412.771,A -85,B 0,C 180,E1 14203.467,E2 14203.467} C_VEL
LIN {X 0,Y 334.466,Z 413.353,A -85,B 0,C 180,E1 14198.794,E2 14198.794} C_VEL
LIN {X 0,Y 337.232,Z 417.753,A -85,B 0,C 180,E1 14192.258,E2 14192.258} C_VEL
LIN {X 0,Y 340.433,Z 419.842,A -85,B 0,C 180,E1 14188.282,E2 14188.282} C_VEL
LIN {X 0,Y 342.727,Z 423.724,A -85,B 0,C 180,E1 14185.732,E2 14185.732} C_VEL
LIN {X 0,Y 346.096,Z 426.333,A -85,B 0,C 180,E1 14182.909,E2 14182.909} C_VEL
LIN {X 0,Y 348.752,Z 430.289,A -85,B 0,C 180,E1 14180.789,E2 14180.789} C_VEL
LIN {X 0,Y 351.591,Z 432.714,A -85,B 0,C 180,E1 14178.895,E2 14178.895} C_VEL
LIN {X 0,Y 354.78,Z 437.028,A -85,B 0,C 180,E1 14176.872,E2 14176.872} C_VEL
LIN {X 0,Y 356.929,Z 439.085,A -85,B 0,C 180,E1 14175.659,E2 14175.659} C_VEL
LIN {X 0,Y 360.475,Z 443.538,A -85,B 0,C 180,E1 14173.733,E2 14173.733} C_VEL
LIN {X 0,Y 362.118,Z 445.35,A -85,B 0,C 180,E1 14172.912,E2 14172.912} C_VEL
LIN {X 0,Y 365.993,Z 449.989,A -85,B 0,C 180,E1 14171.061,E2 14171.061} C_VEL
LIN {X 0,Y 371.934,Z 457.603,A -85,B 0,C 180,E1 14168.461,E2 14168.461} C_VEL
LIN {X 0,Y 376.671,Z 463.612,A -85,B 0,C 180,E1 14166.584,E2 14166.584} C_VEL
LIN {X 0,Y 382.96,Z 471.689,A -85,B 0,C 180,E1 14164.288,E2 14164.288} C_VEL
LIN {X 0,Y 393.147,Z 485.744,A -85,B 0,C 180,E1 14160.933,E2 14160.933} C_VEL
LIN {X 0,Y 401.887,Z 498.543,A -85,B 0,C 180,E1 14158.351,E2 14158.351} C_VEL
LIN {X 0,Y 388.656,Z 705.722,A -85,B 0,C 180,E1 14154.21,E2 14154.21} C_VEL
LIN {X 0,Y 386.551,Z 728.536,A -85,B 0,C 180,E1 14153.661,E2 14153.661} C_VEL
LIN {X 0,Y 383.284,Z 752.483,A -85,B 0,C 180,E1 14152.863,E2 14152.863} C_VEL
LIN {X 0,Y 379.799,Z 772.414,A -85,B 0,C 180,E1 14151.988,E2 14151.988} C_VEL
LIN {X 0,Y 374.962,Z 795.227,A -85,B 0,C 180,E1 14150.717,E2 14150.717} C_VEL
LIN {X 0,Y 370.218,Z 814.48,A -85,B 0,C 180,E1 14149.397,E2 14149.397} C_VEL
LIN {X 0,Y 364.314,Z 835.416,A -85,B 0,C 180,E1 14147.649,E2 14147.649} C_VEL
LIN {X 0,Y 358.375,Z 854.596,A -85,B 0,C 180,E1 14145.73,E2 14145.73} C_VEL
LIN {X 0,Y 352.145,Z 872.718,A -85,B 0,C 180,E1 14143.542,E2 14143.542} C_VEL
LIN {X 0,Y 345.722,Z 890.506,A -85,B 0,C 180,E1 14140.999,E2 14140.999} C_VEL
LIN {X 0,Y 339.671,Z 906.345,A -85,B 0,C 180,E1 14138.288,E2 14138.288} C_VEL
LIN {X 0,Y 333.329,Z 922.566,A -85,B 0,C 180,E1 14134.986,E2 14134.986} C_VEL
LIN {X 0,Y 328.103,Z 936.011,A -85,B 0,C 180,E1 14131.715,E2 14131.715} C_VEL
LIN {X 0,Y 326.075,Z 941.156,A -85,B 0,C 180,E1 14130.277,E2 14130.277} C_VEL
LIN {X 0,Y 323.661,Z 945.261,A -85,B 0,C 180,E1 14129.185,E2 14129.185} C_VEL
LIN {X 0,Y 314.545,Z 955.097,A -85,B 0,C 180,E1 14126.491,E2 14126.491} C_VEL
LIN {X 0,Y 312.366,Z 958.611,A -85,B 0,C 180,E1 14125.292,E2 14125.292} C_VEL
LIN {X 0,Y 309.059,Z 967.961,A -85,B 0,C 180,E1 14121.249,E2 14121.249} C_VEL
LIN {X 0,Y 306.707,Z 975.836,A -85,B 0,C 180,E1 14117.095,E2 14117.095} C_VEL
LIN {X 0,Y 305.241,Z 981.781,A -85,B 0,C 180,E1 14113.037,E2 14113.037} C_VEL
LIN {X 0,Y 304.404,Z 986.512,A -85,B 0,C 180,E1 14108.815,E2 14108.815} C_VEL
LIN {X 0,Y 304.076,Z 989.427,A -85,B 0,C 180,E1 14104.897,E2 14104.897} C_VEL
LIN {X 0,Y 303.998,Z 991.15,A -85,B 0,C 180,E1 14101.032,E2 14101.032} C_VEL
LIN {X 0,Y 303.967,Z 991.518,A -85,B 0,C 180,E1 14096.9,E2 14096.9} C_VEL
LIN {X 0,Y 303.99,Z 990.775,A -85,B 0,C 180,E1 14093.459,E2 14093.459} C_VEL
LIN {X 0,Y 304.183,Z 988.701,A -85,B 0,C 180,E1 14089.391,E2 14089.391} C_VEL
LIN {X 0,Y 304.695,Z 985.179,A -85,B 0,C 180,E1 14085.388,E2 14085.388} C_VEL
LIN {X 0,Y 305.797,Z 980.221,A -85,B 0,C 180,E1 14081.229,E2 14081.229} C_VEL
LIN {X 0,Y 307.65,Z 973.577,A -85,B 0,C 180,E1 14077.089,E2 14077.089} C_VEL
LIN {X 0,Y 310.465,Z 965.444,A -85,B 0,C 180,E1 14072.975,E2 14072.975} C_VEL
LIN {X 0,Y 314.052,Z 956.031,A -85,B 0,C 180,E1 14069.152,E2 14069.152} C_VEL
LIN {X 0,Y 318.873,Z 944.51,A -85,B 0,C 180,E1 14065.243,E2 14065.243} C_VEL
LIN {X 0,Y 324.158,Z 932.261,A -85,B 0,C 180,E1 14061.801,E2 14061.801} C_VEL
LIN {X 0,Y 330.697,Z 917.316,A -85,B 0,C 180,E1 14058.301,E2 14058.301} C_VEL
LIN {X 0,Y 337.356,Z 902.014,A -85,B 0,C 180,E1 14055.295,E2 14055.295} C_VEL
LIN {X 0,Y 344.261,Z 885.337,A -85,B 0,C 180,E1 14052.582,E2 14052.582} C_VEL
LIN {X 0,Y 351.247,Z 867.781,A -85,B 0,C 180,E1 14050.166,E2 14050.166} C_VEL
LIN {X 0,Y 358.096,Z 849.042,A -85,B 0,C 180,E1 14048.026,E2 14048.026} C_VEL
LIN {X 0,Y 365.005,Z 828.335,A -85,B 0,C 180,E1 14046.065,E2 14046.065} C_VEL
LIN {X 0,Y 371.395,Z 807.005,A -85,B 0,C 180,E1 14044.409,E2 14044.409} C_VEL
LIN {X 0,Y 376.753,Z 785.89,A -85,B 0,C 180,E1 14043.094,E2 14043.094} C_VEL
LIN {X 0,Y 381.739,Z 762.94,A -85,B 0,C 180,E1 14041.952,E2 14041.952} C_VEL
LIN {X 0,Y 385.428,Z 741.395,A -85,B 0,C 180,E1 14041.129,E2 14041.129} C_VEL
LIN {X 0,Y 388.548,Z 716.756,A -85,B 0,C 180,E1 14040.447,E2 14040.447} C_VEL
LIN {X 0,Y 406.005,Z 510.781,A -85,B 0,C 180,E1 14036.133,E2 14036.133} C_VEL
LIN {X 0,Y 406.348,Z 506.251,A -85,B 0,C 180,E1 14036.015,E2 14036.015} C_VEL
LIN {X 0,Y 402.16,Z 498.575,A -85,B 0,C 180,E1 14033.828,E2 14033.828} C_VEL
LIN {X 0,Y 399.761,Z 494.329,A -85,B 0,C 180,E1 14032.311,E2 14032.311} C_VEL
LIN {X 0,Y 398.089,Z 491.295,A -85,B 0,C 180,E1 14031.042,E2 14031.042} C_VEL
LIN {X 0,Y 396.076,Z 487.556,A -85,B 0,C 180,E1 14029.087,E2 14029.087} C_VEL
LIN {X 0,Y 394.296,Z 483.864,A -85,B 0,C 180,E1 14025.836,E2 14025.836} C_VEL
LIN {X 0,Y 394.169,Z 483.168,A -85,B 0,C 180,E1 14025.005,E2 14025.005} C_VEL
LIN {X 0,Y 394.25,Z 483.453,A -85,B 0,C 180,E1 14022.892,E2 14022.892} C_VEL
LIN {X 0,Y 395.614,Z 487.027,A -85,B 0,C 180,E1 14019.897,E2 14019.897} C_VEL
LIN {X 0,Y 396.513,Z 488.379,A -85,B 0,C 180,E1 14018.864,E2 14018.864} C_VEL
LIN {X 0,Y 399.009,Z 492.923,A -85,B 0,C 180,E1 14016.677,E2 14016.677} C_VEL
LIN {X 0,Y 401.853,Z 498.856,A -85,B 0,C 180,E1 14014.741,E2 14014.741} C_VEL
LIN {X 0,Y 405.808,Z 507.385,A -85,B 0,C 180,E1 14012.565,E2 14012.565} C_VEL
LIN {X 0,Y 406.306,Z 508.847,A -85,B 0,C 180,E1 14012.305,E2 14012.305} C_VEL
LIN {X 0,Y 390.923,Z 691.222,A -85,B 0,C 180,E1 14008.494,E2 14008.494} C_VEL
LIN {X 0,Y 387.18,Z 735.226,A -85,B 0,C 180,E1 14007.539,E2 14007.539} C_VEL
LIN {X 0,Y 383.801,Z 758.548,A -85,B 0,C 180,E1 14006.875,E2 14006.875} C_VEL
LIN {X 0,Y 379.367,Z 781.842,A -85,B 0,C 180,E1 14005.989,E2 14005.989} C_VEL
LIN {X 0,Y 374.712,Z 802.034,A -85,B 0,C 180,E1 14004.993,E2 14004.993} C_VEL
LIN {X 0,Y 368.834,Z 824.132,A -85,B 0,C 180,E1 14003.627,E2 14003.627} C_VEL
LIN {X 0,Y 362.88,Z 843.91,A -85,B 0,C 180,E1 14002.121,E2 14002.121} C_VEL
LIN {X 0,Y 355.929,Z 864.743,A -85,B 0,C 180,E1 14000.193,E2 14000.193} C_VEL
LIN {X 0,Y 348.979,Z 884.136,A -85,B 0,C 180,E1 13998.034,E2 13998.034} C_VEL
LIN {X 0,Y 341.819,Z 902.599,A -85,B 0,C 180,E1 13995.543,E2 13995.543} C_VEL
LIN {X 0,Y 334.566,Z 920.816,A -85,B 0,C 180,E1 13992.606,E2 13992.606} C_VEL
LIN {X 0,Y 328.46,Z 935.743,A -85,B 0,C 180,E1 13989.741,E2 13989.741} C_VEL
LIN {X 0,Y 322.149,Z 951.251,A -85,B 0,C 180,E1 13986.201,E2 13986.201} C_VEL
LIN {X 0,Y 316.762,Z 965.015,A -85,B 0,C 180,E1 13982.457,E2 13982.457} C_VEL
LIN {X 0,Y 312.316,Z 976.978,A -85,B 0,C 180,E1 13978.495,E2 13978.495} C_VEL
LIN {X 0,Y 308.837,Z 987.571,A -85,B 0,C 180,E1 13974.282,E2 13974.282} C_VEL
LIN {X 0,Y 306.626,Z 995.499,A -85,B 0,C 180,E1 13970.425,E2 13970.425} C_VEL
LIN {X 0,Y 305.028,Z 1002.81,A -85,B 0,C 180,E1 13965.987,E2 13965.987} C_VEL
LIN {X 0,Y 304.325,Z 1007.446,A -85,B 0,C 180,E1 13962.336,E2 13962.336} C_VEL
LIN {X 0,Y 304.017,Z 1011.361,A -85,B 0,C 180,E1 13958.135,E2 13958.135} C_VEL
LIN {X 0,Y 303.956,Z 1013.456,A -85,B 0,C 180,E1 13954.344,E2 13954.344} C_VEL
LIN {X 0,Y 303.957,Z 1014.299,A -85,B 0,C 180,E1 13950.947,E2 13950.947} C_VEL
LIN {X 0,Y 303.944,Z 1014,A -85,B 0,C 180,E1 13946.988,E2 13946.988} C_VEL
LIN {X 0,Y 303.972,Z 1012.417,A -85,B 0,C 180,E1 13943.394,E2 13943.394} C_VEL
LIN {X 0,Y 304.091,Z 1009.883,A -85,B 0,C 180,E1 13939.969,E2 13939.969} C_VEL
LIN {X 0,Y 304.64,Z 1005.372,A -85,B 0,C 180,E1 13935.755,E2 13935.755} C_VEL
LIN {X 0,Y 305.674,Z 999.736,A -85,B 0,C 180,E1 13931.902,E2 13931.902} C_VEL
LIN {X 0,Y 307.517,Z 992.385,A -85,B 0,C 180,E1 13927.848,E2 13927.848} C_VEL
LIN {X 0,Y 310.281,Z 983.168,A -85,B 0,C 180,E1 13923.809,E2 13923.809} C_VEL
LIN {X 0,Y 314.088,Z 972.198,A -85,B 0,C 180,E1 13919.81,E2 13919.81} C_VEL
LIN {X 0,Y 318.484,Z 960.415,A -85,B 0,C 180,E1 13916.25,E2 13916.25} C_VEL
LIN {X 0,Y 324.129,Z 945.93,A -85,B 0,C 180,E1 13912.584,E2 13912.584} C_VEL
LIN {X 0,Y 330.143,Z 930.837,A -85,B 0,C 180,E1 13909.38,E2 13909.38} C_VEL
LIN {X 0,Y 336.58,Z 914.213,A -85,B 0,C 180,E1 13906.442,E2 13906.442} C_VEL
LIN {X 0,Y 343.372,Z 896.264,A -85,B 0,C 180,E1 13903.777,E2 13903.777} C_VEL
LIN {X 0,Y 349.62,Z 878.641,A -85,B 0,C 180,E1 13901.592,E2 13901.592} C_VEL
LIN {X 0,Y 356.532,Z 857.671,A -85,B 0,C 180,E1 13899.42,E2 13899.42} C_VEL
LIN {X 0,Y 362.269,Z 838.591,A -85,B 0,C 180,E1 13897.786,E2 13897.786} C_VEL
LIN {X 0,Y 367.821,Z 817.712,A -85,B 0,C 180,E1 13896.317,E2 13896.317} C_VEL
LIN {X 0,Y 372.75,Z 796.59,A -85,B 0,C 180,E1 13895.112,E2 13895.112} C_VEL
LIN {X 0,Y 377.147,Z 773.666,A -85,B 0,C 180,E1 13894.094,E2 13894.094} C_VEL
LIN {X 0,Y 380.757,Z 750.494,A -85,B 0,C 180,E1 13893.32,E2 13893.32} C_VEL
LIN {X 0,Y 383.114,Z 727.397,A -85,B 0,C 180,E1 13892.755,E2 13892.755} C_VEL
LIN {X 0,Y 396.978,Z 517.895,A -85,B 0,C 180,E1 13888.533,E2 13888.533} C_VEL
LIN {X 0,Y 397.677,Z 506.613,A -85,B 0,C 180,E1 13888.29,E2 13888.29} C_VEL
LIN {X 0,Y 389.209,Z 492.898,A -85,B 0,C 180,E1 13885.649,E2 13885.649} C_VEL
LIN {X 0,Y 381.262,Z 480.741,A -85,B 0,C 180,E1 13882.919,E2 13882.919} C_VEL
LIN {X 0,Y 372.609,Z 468.345,A -85,B 0,C 180,E1 13879.598,E2 13879.598} C_VEL
LIN {X 0,Y 367.081,Z 461.556,A -85,B 0,C 180,E1 13877.271,E2 13877.271} C_VEL
LIN {X 0,Y 363.392,Z 456.842,A -85,B 0,C 180,E1 13875.561,E2 13875.561} C_VEL
LIN {X 0,Y 359.153,Z 451.53,A -85,B 0,C 180,E1 13873.441,E2 13873.441} C_VEL
LIN {X 0,Y 355.385,Z 447.08,A -85,B 0,C 180,E1 13871.399,E2 13871.399} C_VEL
LIN {X 0,Y 354.262,Z 445.687,A -85,B 0,C 180,E1 13870.735,E2 13870.735} C_VEL
LIN {X 0,Y 350.672,Z 441.613,A -85,B 0,C 180,E1 13868.526,E2 13868.526} C_VEL
LIN {X 0,Y 349.535,Z 439.885,A -85,B 0,C 180,E1 13867.726,E2 13867.726} C_VEL
LIN {X 0,Y 346.092,Z 436.632,A -85,B 0,C 180,E1 13865.304,E2 13865.304} C_VEL
LIN {X 0,Y 344.161,Z 433.599,A -85,B 0,C 180,E1 13863.664,E2 13863.664} C_VEL
LIN {X 0,Y 340.862,Z 430.931,A -85,B 0,C 180,E1 13860.756,E2 13860.756} C_VEL
LIN {X 0,Y 338.778,Z 427.263,A -85,B 0,C 180,E1 13858.308,E2 13858.308} C_VEL
LIN {X 0,Y 335.167,Z 424.763,A -85,B 0,C 180,E1 13853.318,E2 13853.318} C_VEL
LIN {X 0,Y 333.313,Z 421.274,A -85,B 0,C 180,E1 13848.229,E2 13848.229} C_VEL
LIN {X 0,Y 332.698,Z 420.693,A -85,B 0,C 180,E1 13843.452,E2 13843.452} C_VEL
LIN {X 0,Y 333.376,Z 421.313,A -85,B 0,C 180,E1 13838.721,E2 13838.721} C_VEL
LIN {X 0,Y 336.06,Z 425.652,A -85,B 0,C 180,E1 13832.345,E2 13832.345} C_VEL
LIN {X 0,Y 339.077,Z 427.615,A -85,B 0,C 180,E1 13828.538,E2 13828.538} C_VEL
LIN {X 0,Y 341.438,Z 431.568,A -85,B 0,C 180,E1 13825.889,E2 13825.889} C_VEL
LIN {X 0,Y 344.595,Z 434.05,A -85,B 0,C 180,E1 13823.199,E2 13823.199} C_VEL
LIN {X 0,Y 347.406,Z 438.161,A -85,B 0,C 180,E1 13820.927,E2 13820.927} C_VEL
LIN {X 0,Y 350.042,Z 440.515,A -85,B 0,C 180,E1 13819.147,E2 13819.147} C_VEL
LIN {X 0,Y 353.389,Z 444.899,A -85,B 0,C 180,E1 13817.009,E2 13817.009} C_VEL
LIN {X 0,Y 355.217,Z 446.757,A -85,B 0,C 180,E1 13815.952,E2 13815.952} C_VEL
LIN {X 0,Y 358.959,Z 451.344,A -85,B 0,C 180,E1 13813.906,E2 13813.906} C_VEL
LIN {X 0,Y 360.691,Z 453.548,A -85,B 0,C 180,E1 13813.012,E2 13813.012} C_VEL
LIN {X 0,Y 365.009,Z 458.836,A -85,B 0,C 180,E1 13810.943,E2 13810.943} C_VEL
LIN {X 0,Y 369.785,Z 464.906,A -85,B 0,C 180,E1 13808.845,E2 13808.845} C_VEL
LIN {X 0,Y 374.575,Z 471.078,A -85,B 0,C 180,E1 13806.906,E2 13806.906} C_VEL
LIN {X 0,Y 380.554,Z 478.908,A -85,B 0,C 180,E1 13804.677,E2 13804.677} C_VEL
LIN {X 0,Y 390.336,Z 492.56,A -85,B 0,C 180,E1 13801.39,E2 13801.39} C_VEL
LIN {X 0,Y 397.369,Z 503.226,A -85,B 0,C 180,E1 13799.239,E2 13799.239} C_VEL
LIN {X 0,Y 383.498,Z 711.275,A -85,B 0,C 180,E1 13795.051,E2 13795.051} C_VEL
LIN {X 0,Y 381.051,Z 734.796,A -85,B 0,C 180,E1 13794.447,E2 13794.447} C_VEL
LIN {X 0,Y 377.758,Z 756.565,A -85,B 0,C 180,E1 13793.666,E2 13793.666} C_VEL
LIN {X 0,Y 373.684,Z 778.382,A -85,B 0,C 180,E1 13792.657,E2 13792.657} C_VEL
LIN {X 0,Y 369,Z 798.966,A -85,B 0,C 180,E1 13791.452,E2 13791.452} C_VEL
LIN {X 0,Y 363.27,Z 820.725,A -85,B 0,C 180,E1 13789.885,E2 13789.885} C_VEL
LIN {X 0,Y 357.661,Z 839.488,A -85,B 0,C 180,E1 13788.241,E2 13788.241} C_VEL
LIN {X 0,Y 351.003,Z 859.601,A -85,B 0,C 180,E1 13786.12,E2 13786.12} C_VEL
LIN {X 0,Y 344.527,Z 877.765,A -85,B 0,C 180,E1 13783.829,E2 13783.829} C_VEL
LIN {X 0,Y 338.007,Z 894.72,A -85,B 0,C 180,E1 13781.253,E2 13781.253} C_VEL
LIN {X 0,Y 331.849,Z 910.226,A -85,B 0,C 180,E1 13778.485,E2 13778.485} C_VEL
LIN {X 0,Y 325.679,Z 925.143,A -85,B 0,C 180,E1 13775.28,E2 13775.28} C_VEL
LIN {X 0,Y 319.834,Z 939.44,A -85,B 0,C 180,E1 13771.608,E2 13771.608} C_VEL
LIN {X 0,Y 315.405,Z 950.57,A -85,B 0,C 180,E1 13768.179,E2 13768.179} C_VEL
LIN {X 0,Y 312.366,Z 958.611,A -85,B 0,C 180,E1 13765.292,E2 13765.292} C_VEL
LIN {X 0,Y 310.266,Z 961.995,A -85,B 0,C 180,E1 13764.066,E2 13764.066} C_VEL
LIN {X 0,Y 301.507,Z 970.286,A -85,B 0,C 180,E1 13760.782,E2 13760.782} C_VEL
LIN {X 0,Y 300.019,Z 972.536,A -85,B 0,C 180,E1 13759.619,E2 13759.619} C_VEL
LIN {X 0,Y 298.084,Z 979.098,A -85,B 0,C 180,E1 13755.623,E2 13755.623} C_VEL
LIN {X 0,Y 296.797,Z 984.74,A -85,B 0,C 180,E1 13751.126,E2 13751.126} C_VEL
LIN {X 0,Y 296.245,Z 988.19,A -85,B 0,C 180,E1 13747.366,E2 13747.366} C_VEL
LIN {X 0,Y 296.011,Z 990.747,A -85,B 0,C 180,E1 13743.083,E2 13743.083} C_VEL
LIN {X 0,Y 295.969,Z 991.726,A -85,B 0,C 180,E1 13739.481,E2 13739.481} C_VEL
LIN {X 0,Y 295.966,Z 991.722,A -85,B 0,C 180,E1 13735.862,E2 13735.862} C_VEL
LIN {X 0,Y 296.049,Z 990.522,A -85,B 0,C 180,E1 13731.821,E2 13731.821} C_VEL
LIN {X 0,Y 296.362,Z 987.983,A -85,B 0,C 180,E1 13727.821,E2 13727.821} C_VEL
LIN {X 0,Y 297.098,Z 984.085,A -85,B 0,C 180,E1 13723.624,E2 13723.624} C_VEL
LIN {X 0,Y 298.6,Z 978.341,A -85,B 0,C 180,E1 13719.262,E2 13719.262} C_VEL
LIN {X 0,Y 301.061,Z 971.003,A -85,B 0,C 180,E1 13714.878,E2 13714.878} C_VEL
LIN {X 0,Y 304.519,Z 962.014,A -85,B 0,C 180,E1 13710.649,E2 13710.649} C_VEL
LIN {X 0,Y 309.25,Z 950.945,A -85,B 0,C 180,E1 13706.409,E2 13706.409} C_VEL
LIN {X 0,Y 314.739,Z 938.926,A -85,B 0,C 180,E1 13702.607,E2 13702.607} C_VEL
LIN {X 0,Y 320.915,Z 925.415,A -85,B 0,C 180,E1 13699.096,E2 13699.096} C_VEL
LIN {X 0,Y 327.815,Z 910.495,A -85,B 0,C 180,E1 13695.842,E2 13695.842} C_VEL
LIN {X 0,Y 334.625,Z 895.195,A -85,B 0,C 180,E1 13693.061,E2 13693.061} C_VEL
LIN {X 0,Y 342.503,Z 876.703,A -85,B 0,C 180,E1 13690.258,E2 13690.258} C_VEL
LIN {X 0,Y 349.493,Z 859.297,A -85,B 0,C 180,E1 13688.059,E2 13688.059} C_VEL
LIN {X 0,Y 356.55,Z 840.004,A -85,B 0,C 180,E1 13686.037,E2 13686.037} C_VEL
LIN {X 0,Y 363.007,Z 820.728,A -85,B 0,C 180,E1 13684.349,E2 13684.349} C_VEL
LIN {X 0,Y 369.023,Z 800.06,A -85,B 0,C 180,E1 13682.874,E2 13682.874} C_VEL
LIN {X 0,Y 374.402,Z 779.011,A -85,B 0,C 180,E1 13681.646,E2 13681.646} C_VEL
LIN {X 0,Y 378.867,Z 757.573,A -85,B 0,C 180,E1 13680.664,E2 13680.664} C_VEL
LIN {X 0,Y 382.68,Z 734.907,A -85,B 0,C 180,E1 13679.865,E2 13679.865} C_VEL
LIN {X 0,Y 385.285,Z 712.838,A -85,B 0,C 180,E1 13679.298,E2 13679.298} C_VEL
LIN {X 0,Y 402.548,Z 518.036,A -85,B 0,C 180,E1 13675.214,E2 13675.214} C_VEL
LIN {X 0,Y 403.141,Z 511.324,A -85,B 0,C 180,E1 13675.056,E2 13675.056} C_VEL
LIN {X 0,Y 399.684,Z 504.747,A -85,B 0,C 180,E1 13673.068,E2 13673.068} C_VEL
LIN {X 0,Y 396.613,Z 498.96,A -85,B 0,C 180,E1 13670.789,E2 13670.789} C_VEL
LIN {X 0,Y 394.78,Z 495.356,A -85,B 0,C 180,E1 13668.903,E2 13668.903} C_VEL
LIN {X 0,Y 393.132,Z 491.755,A -85,B 0,C 180,E1 13665.704,E2 13665.704} C_VEL
LIN {X 0,Y 393.043,Z 491.084,A -85,B 0,C 180,E1 13664.961,E2 13664.961} C_VEL
LIN {X 0,Y 393.103,Z 491.39,A -85,B 0,C 180,E1 13662.993,E2 13662.993} C_VEL
LIN {X 0,Y 394.401,Z 494.918,A -85,B 0,C 180,E1 13659.987,E2 13659.987} C_VEL
LIN {X 0,Y 395.144,Z 496.12,A -85,B 0,C 180,E1 13659.098,E2 13659.098} C_VEL
LIN {X 0,Y 397.441,Z 500.517,A -85,B 0,C 180,E1 13656.972,E2 13656.972} C_VEL
LIN {X 0,Y 400.135,Z 506.536,A -85,B 0,C 180,E1 13655.021,E2 13655.021} C_VEL
LIN {X 0,Y 403.122,Z 513.283,A -85,B 0,C 180,E1 13653.282,E2 13653.282} C_VEL
LIN {X 0,Y 387.062,Z 694.697,A -85,B 0,C 180,E1 13649.48,E2 13649.48} C_VEL
LIN {X 0,Y 383.311,Z 735.884,A -85,B 0,C 180,E1 13648.576,E2 13648.576} C_VEL
LIN {X 0,Y 379.844,Z 758.764,A -85,B 0,C 180,E1 13647.922,E2 13647.922} C_VEL
LIN {X 0,Y 375.154,Z 782.245,A -85,B 0,C 180,E1 13647.025,E2 13647.025} C_VEL
LIN {X 0,Y 369.932,Z 804.032,A -85,B 0,C 180,E1 13645.94,E2 13645.94} C_VEL
LIN {X 0,Y 364.124,Z 824.631,A -85,B 0,C 180,E1 13644.645,E2 13644.645} C_VEL
LIN {X 0,Y 357.441,Z 845.971,A -85,B 0,C 180,E1 13643.003,E2 13643.003} C_VEL
LIN {X 0,Y 350.519,Z 865.543,A -85,B 0,C 180,E1 13641.149,E2 13641.149} C_VEL
LIN {X 0,Y 343.286,Z 884.786,A -85,B 0,C 180,E1 13638.974,E2 13638.974} C_VEL
LIN {X 0,Y 335.844,Z 903.101,A -85,B 0,C 180,E1 13636.468,E2 13636.468} C_VEL
LIN {X 0,Y 328.068,Z 921.605,A -85,B 0,C 180,E1 13633.418,E2 13633.418} C_VEL
LIN {X 0,Y 321.357,Z 937.289,A -85,B 0,C 180,E1 13630.332,E2 13630.332} C_VEL
LIN {X 0,Y 315.025,Z 951.933,A -85,B 0,C 180,E1 13626.865,E2 13626.865} C_VEL
LIN {X 0,Y 309.457,Z 965.341,A -85,B 0,C 180,E1 13623.1,E2 13623.1} C_VEL
LIN {X 0,Y 304.982,Z 976.7,A -85,B 0,C 180,E1 13619.245,E2 13619.245} C_VEL
LIN {X 0,Y 301.116,Z 987.696,A -85,B 0,C 180,E1 13614.737,E2 13614.737} C_VEL
LIN {X 0,Y 298.774,Z 995.572,A -85,B 0,C 180,E1 13610.782,E2 13610.782} C_VEL
LIN {X 0,Y 297.087,Z 1002.775,A -85,B 0,C 180,E1 13606.225,E2 13606.225} C_VEL
LIN {X 0,Y 296.314,Z 1007.582,A -85,B 0,C 180,E1 13602.278,E2 13602.278} C_VEL
LIN {X 0,Y 296.008,Z 1011.304,A -85,B 0,C 180,E1 13597.965,E2 13597.965} C_VEL
LIN {X 0,Y 295.961,Z 1013.232,A -85,B 0,C 180,E1 13594.267,E2 13594.267} C_VEL
LIN {X 0,Y 295.963,Z 1014.074,A -85,B 0,C 180,E1 13590.424,E2 13590.424} C_VEL
LIN {X 0,Y 295.951,Z 1013.557,A -85,B 0,C 180,E1 13586.519,E2 13586.519} C_VEL
LIN {X 0,Y 295.964,Z 1011.99,A -85,B 0,C 180,E1 13583.02,E2 13583.02} C_VEL
LIN {X 0,Y 296.125,Z 1009.4,A -85,B 0,C 180,E1 13579.5,E2 13579.5} C_VEL
LIN {X 0,Y 296.745,Z 1004.771,A -85,B 0,C 180,E1 13575.168,E2 13575.168} C_VEL
LIN {X 0,Y 297.912,Z 999.067,A -85,B 0,C 180,E1 13571.21,E2 13571.21} C_VEL
LIN {X 0,Y 300.08,Z 991.168,A -85,B 0,C 180,E1 13566.854,E2 13566.854} C_VEL
LIN {X 0,Y 302.975,Z 982.297,A -85,B 0,C 180,E1 13562.915,E2 13562.915} C_VEL
LIN {X 0,Y 307.305,Z 970.568,A -85,B 0,C 180,E1 13558.636,E2 13558.636} C_VEL
LIN {X 0,Y 312.337,Z 957.966,A -85,B 0,C 180,E1 13554.822,E2 13554.822} C_VEL
LIN {X 0,Y 318.142,Z 943.818,A -85,B 0,C 180,E1 13551.295,E2 13551.295} C_VEL
LIN {X 0,Y 324.539,Z 928.393,A -85,B 0,C 180,E1 13548.053,E2 13548.053} C_VEL
LIN {X 0,Y 330.969,Z 912.506,A -85,B 0,C 180,E1 13545.268,E2 13545.268} C_VEL
LIN {X 0,Y 338.415,Z 893.384,A -85,B 0,C 180,E1 13542.467,E2 13542.467} C_VEL
LIN {X 0,Y 345.061,Z 875.283,A -85,B 0,C 180,E1 13540.253,E2 13540.253} C_VEL
LIN {X 0,Y 351.559,Z 855.894,A -85,B 0,C 180,E1 13538.292,E2 13538.292} C_VEL
LIN {X 0,Y 357.869,Z 835.444,A -85,B 0,C 180,E1 13536.568,E2 13536.568} C_VEL
LIN {X 0,Y 363.624,Z 813.913,A -85,B 0,C 180,E1 13535.108,E2 13535.108} C_VEL
LIN {X 0,Y 369.11,Z 790.174,A -85,B 0,C 180,E1 13533.827,E2 13533.827} C_VEL
LIN {X 0,Y 373.207,Z 768.68,A -85,B 0,C 180,E1 13532.927,E2 13532.927} C_VEL
LIN {X 0,Y 376.678,Z 745.072,A -85,B 0,C 180,E1 13532.198,E2 13532.198} C_VEL
LIN {X 0,Y 378.962,Z 721.105,A -85,B 0,C 180,E1 13531.635,E2 13531.635} C_VEL
LIN {X 0,Y 393.072,Z 514.149,A -85,B 0,C 180,E1 13527.462,E2 13527.462} C_VEL
LIN {X 0,Y 393.199,Z 510.698,A -85,B 0,C 180,E1 13527.362,E2 13527.362} C_VEL
LIN {X 0,Y 383.46,Z 494.963,A -85,B 0,C 180,E1 13524.165,E2 13524.165} C_VEL
LIN {X 0,Y 375.281,Z 482.602,A -85,B 0,C 180,E1 13521.162,E2 13521.162} C_VEL
LIN {X 0,Y 369.3,Z 474.358,A -85,B 0,C 180,E1 13518.754,E2 13518.754} C_VEL
LIN {X 0,Y 365.146,Z 469.057,A -85,B 0,C 180,E1 13516.955,E2 13516.955} C_VEL
LIN {X 0,Y 361.166,Z 464.003,A -85,B 0,C 180,E1 13515.083,E2 13515.083} C_VEL
LIN {X 0,Y 357.156,Z 458.905,A -85,B 0,C 180,E1 13513.023,E2 13513.023} C_VEL
LIN {X 0,Y 353.409,Z 454.266,A -85,B 0,C 180,E1 13510.926,E2 13510.926} C_VEL
LIN {X 0,Y 348.844,Z 448.903,A -85,B 0,C 180,E1 13508.073,E2 13508.073} C_VEL
LIN {X 0,Y 347.731,Z 447.434,A -85,B 0,C 180,E1 13507.3,E2 13507.3} C_VEL
LIN {X 0,Y 344.252,Z 443.832,A -85,B 0,C 180,E1 13504.748,E2 13504.748} C_VEL
LIN {X 0,Y 342.837,Z 441.442,A -85,B 0,C 180,E1 13503.511,E2 13503.511} C_VEL
LIN {X 0,Y 339.488,Z 438.671,A -85,B 0,C 180,E1 13500.506,E2 13500.506} C_VEL
LIN {X 0,Y 337.502,Z 435.122,A -85,B 0,C 180,E1 13498.132,E2 13498.132} C_VEL
LIN {X 0,Y 333.939,Z 432.594,A -85,B 0,C 180,E1 13493.121,E2 13493.121} C_VEL
LIN {X 0,Y 332.14,Z 429.147,A -85,B 0,C 180,E1 13488.011,E2 13488.011} C_VEL
LIN {X 0,Y 331.599,Z 428.601,A -85,B 0,C 180,E1 13483.174,E2 13483.174} C_VEL
LIN {X 0,Y 332.282,Z 429.309,A -85,B 0,C 180,E1 13478.647,E2 13478.647} C_VEL
LIN {X 0,Y 334.888,Z 433.552,A -85,B 0,C 180,E1 13472.433,E2 13472.433} C_VEL
LIN {X 0,Y 337.728,Z 435.38,A -85,B 0,C 180,E1 13468.795,E2 13468.795} C_VEL
LIN {X 0,Y 340.141,Z 439.412,A -85,B 0,C 180,E1 13466.046,E2 13466.046} C_VEL
LIN {X 0,Y 343.155,Z 441.894,A -85,B 0,C 180,E1 13463.426,E2 13463.426} C_VEL
LIN {X 0,Y 346.2,Z 446.166,A -85,B 0,C 180,E1 13460.968,E2 13460.968} C_VEL
LIN {X 0,Y 348.41,Z 448.133,A -85,B 0,C 180,E1 13459.468,E2 13459.468} C_VEL
LIN {X 0,Y 351.872,Z 452.646,A -85,B 0,C 180,E1 13457.224,E2 13457.224} C_VEL
LIN {X 0,Y 353.516,Z 454.415,A -85,B 0,C 180,E1 13456.248,E2 13456.248} C_VEL
LIN {X 0,Y 357.342,Z 459.05,A -85,B 0,C 180,E1 13454.135,E2 13454.135} C_VEL
LIN {X 0,Y 363.202,Z 466.526,A -85,B 0,C 180,E1 13451.215,E2 13451.215} C_VEL
LIN {X 0,Y 367.815,Z 472.446,A -85,B 0,C 180,E1 13449.157,E2 13449.157} C_VEL
LIN {X 0,Y 374.6,Z 481.184,A -85,B 0,C 180,E1 13446.414,E2 13446.414} C_VEL
LIN {X 0,Y 384.848,Z 495.446,A -85,B 0,C 180,E1 13442.74,E2 13442.74} C_VEL
LIN {X 0,Y 392.936,Z 507.592,A -85,B 0,C 180,E1 13440.15,E2 13440.15} C_VEL
LIN {X 0,Y 378.7,Z 713.458,A -85,B 0,C 180,E1 13435.989,E2 13435.989} C_VEL
LIN {X 0,Y 375.874,Z 738.14,A -85,B 0,C 180,E1 13435.327,E2 13435.327} C_VEL
LIN {X 0,Y 372.545,Z 759.168,A -85,B 0,C 180,E1 13434.55,E2 13434.55} C_VEL
LIN {X 0,Y 367.973,Z 782.029,A -85,B 0,C 180,E1 13433.452,E2 13433.452} C_VEL
LIN {X 0,Y 362.926,Z 803.263,A -85,B 0,C 180,E1 13432.169,E2 13432.169} C_VEL
LIN {X 0,Y 357.226,Z 823.612,A -85,B 0,C 180,E1 13430.645,E2 13430.645} C_VEL
LIN {X 0,Y 351.045,Z 843.509,A -85,B 0,C 180,E1 13428.856,E2 13428.856} C_VEL
LIN {X 0,Y 344.44,Z 862.401,A -85,B 0,C 180,E1 13426.783,E2 13426.783} C_VEL
LIN {X 0,Y 337.505,Z 880.89,A -85,B 0,C 180,E1 13424.363,E2 13424.363} C_VEL
LIN {X 0,Y 331.059,Z 896.953,A -85,B 0,C 180,E1 13421.846,E2 13421.846} C_VEL
LIN {X 0,Y 323.98,Z 913.823,A -85,B 0,C 180,E1 13418.693,E2 13418.693} C_VEL
LIN {X 0,Y 317.742,Z 928.466,A -85,B 0,C 180,E1 13415.412,E2 13415.412} C_VEL
LIN {X 0,Y 312.031,Z 941.641,A -85,B 0,C 180,E1 13411.831,E2 13411.831} C_VEL
LIN {X 0,Y 307.073,Z 953.614,A -85,B 0,C 180,E1 13407.943,E2 13407.943} C_VEL
LIN {X 0,Y 303.283,Z 963.254,A -85,B 0,C 180,E1 13404.129,E2 13404.129} C_VEL
LIN {X 0,Y 300.019,Z 972.536,A -85,B 0,C 180,E1 13399.619,E2 13399.619} C_VEL
LIN {X 0,Y 298.26,Z 975.139,A -85,B 0,C 180,E1 13398.253,E2 13398.253} C_VEL
LIN {X 0,Y 290.481,Z 981.327,A -85,B 0,C 180,E1 13394.592,E2 13394.592} C_VEL
LIN {X 0,Y 289.354,Z 982.949,A -85,B 0,C 180,E1 13393.335,E2 13393.335} C_VEL
LIN {X 0,Y 288.405,Z 987.654,A -85,B 0,C 180,E1 13388.648,E2 13388.648} C_VEL
LIN {X 0,Y 288.081,Z 990.303,A -85,B 0,C 180,E1 13384.724,E2 13384.724} C_VEL
LIN {X 0,Y 287.987,Z 991.908,A -85,B 0,C 180,E1 13380.457,E2 13380.457} C_VEL
LIN {X 0,Y 287.976,Z 992.116,A -85,B 0,C 180,E1 13376.726,E2 13376.726} C_VEL
LIN {X 0,Y 288.016,Z 991.362,A -85,B 0,C 180,E1 13373.084,E2 13373.084} C_VEL
LIN {X 0,Y 288.253,Z 989.247,A -85,B 0,C 180,E1 13368.767,E2 13368.767} C_VEL
LIN {X 0,Y 288.906,Z 985.695,A -85,B 0,C 180,E1 13364.521,E2 13364.521} C_VEL
LIN {X 0,Y 290.26,Z 980.667,A -85,B 0,C 180,E1 13360.103,E2 13360.103} C_VEL
LIN {X 0,Y 292.475,Z 974.037,A -85,B 0,C 180,E1 13355.774,E2 13355.774} C_VEL
LIN {X 0,Y 295.849,Z 965.652,A -85,B 0,C 180,E1 13351.364,E2 13351.364} C_VEL
LIN {X 0,Y 300.206,Z 955.801,A -85,B 0,C 180,E1 13347.212,E2 13347.212} C_VEL
LIN {X 0,Y 305.814,Z 943.912,A -85,B 0,C 180,E1 13343.101,E2 13343.101} C_VEL
LIN {X 0,Y 312.241,Z 930.821,A -85,B 0,C 180,E1 13339.356,E2 13339.356} C_VEL
LIN {X 0,Y 319.264,Z 916.271,A -85,B 0,C 180,E1 13335.951,E2 13335.951} C_VEL
LIN {X 0,Y 326.668,Z 900.779,A -85,B 0,C 180,E1 13332.912,E2 13332.912} C_VEL
LIN {X 0,Y 334.24,Z 884.089,A -85,B 0,C 180,E1 13330.19,E2 13330.19} C_VEL
LIN {X 0,Y 342.271,Z 865.262,A -85,B 0,C 180,E1 13327.647,E2 13327.647} C_VEL
LIN {X 0,Y 349.616,Z 846.771,A -85,B 0,C 180,E1 13325.572,E2 13325.572} C_VEL
LIN {X 0,Y 356.717,Z 826.753,A -85,B 0,C 180,E1 13323.726,E2 13323.726} C_VEL
LIN {X 0,Y 363.385,Z 805.798,A -85,B 0,C 180,E1 13322.137,E2 13322.137} C_VEL
LIN {X 0,Y 368.734,Z 786.25,A -85,B 0,C 180,E1 13320.933,E2 13320.933} C_VEL
LIN {X 0,Y 373.986,Z 763.715,A -85,B 0,C 180,E1 13319.821,E2 13319.821} C_VEL
LIN {X 0,Y 377.963,Z 742.25,A -85,B 0,C 180,E1 13319.004,E2 13319.004} C_VEL
LIN {X 0,Y 381.344,Z 717.723,A -85,B 0,C 180,E1 13318.324,E2 13318.324} C_VEL
LIN {X 0,Y 400.127,Z 516.567,A -85,B 0,C 180,E1 13314.095,E2 13314.095} C_VEL
LIN {X 0,Y 396.984,Z 510.236,A -85,B 0,C 180,E1 13312.038,E2 13312.038} C_VEL
LIN {X 0,Y 394.892,Z 506.217,A -85,B 0,C 180,E1 13310.307,E2 13310.307} C_VEL
LIN {X 0,Y 393.362,Z 503.013,A -85,B 0,C 180,E1 13308.565,E2 13308.565} C_VEL
LIN {X 0,Y 391.947,Z 499.366,A -85,B 0,C 180,E1 13305.372,E2 13305.372} C_VEL
LIN {X 0,Y 391.862,Z 498.935,A -85,B 0,C 180,E1 13304.005,E2 13304.005} C_VEL
LIN {X 0,Y 391.956,Z 499.373,A -85,B 0,C 180,E1 13303.065,E2 13303.065} C_VEL
LIN {X 0,Y 393.314,Z 502.955,A -85,B 0,C 180,E1 13299.929,E2 13299.929} C_VEL
LIN {X 0,Y 394.65,Z 505.775,A -85,B 0,C 180,E1 13298.377,E2 13298.377} C_VEL
LIN {X 0,Y 396.056,Z 508.487,A -85,B 0,C 180,E1 13297.122,E2 13297.122} C_VEL
LIN {X 0,Y 398.89,Z 515.169,A -85,B 0,C 180,E1 13295.017,E2 13295.017} C_VEL
LIN {X 0,Y 400.08,Z 518.263,A -85,B 0,C 180,E1 13294.265,E2 13294.265} C_VEL
LIN {X 0,Y 383.186,Z 700.273,A -85,B 0,C 180,E1 13290.445,E2 13290.445} C_VEL
LIN {X 0,Y 379.724,Z 735.954,A -85,B 0,C 180,E1 13289.655,E2 13289.655} C_VEL
LIN {X 0,Y 376.118,Z 758.762,A -85,B 0,C 180,E1 13289.003,E2 13289.003} C_VEL
LIN {X 0,Y 371.299,Z 781.955,A -85,B 0,C 180,E1 13288.122,E2 13288.122} C_VEL
LIN {X 0,Y 366.001,Z 803.27,A -85,B 0,C 180,E1 13287.069,E2 13287.069} C_VEL
LIN {X 0,Y 359.851,Z 824.271,A -85,B 0,C 180,E1 13285.757,E2 13285.757} C_VEL
LIN {X 0,Y 353.218,Z 844.655,A -85,B 0,C 180,E1 13284.198,E2 13284.198} C_VEL
LIN {X 0,Y 345.748,Z 865.056,A -85,B 0,C 180,E1 13282.277,E2 13282.277} C_VEL
LIN {X 0,Y 338.178,Z 884.341,A -85,B 0,C 180,E1 13280.091,E2 13280.091} C_VEL
LIN {X 0,Y 330.451,Z 902.541,A -85,B 0,C 180,E1 13277.59,E2 13277.59} C_VEL
LIN {X 0,Y 322.282,Z 921.036,A -85,B 0,C 180,E1 13274.524,E2 13274.524} C_VEL
LIN {X 0,Y 315.412,Z 936.266,A -85,B 0,C 180,E1 13271.498,E2 13271.498} C_VEL
LIN {X 0,Y 308.677,Z 951.008,A -85,B 0,C 180,E1 13267.989,E2 13267.989} C_VEL
LIN {X 0,Y 302.744,Z 964.505,A -85,B 0,C 180,E1 13264.161,E2 13264.161} C_VEL
LIN {X 0,Y 297.911,Z 975.902,A -85,B 0,C 180,E1 13260.232,E2 13260.232} C_VEL
LIN {X 0,Y 293.864,Z 986.571,A -85,B 0,C 180,E1 13255.823,E2 13255.823} C_VEL
LIN {X 0,Y 291.239,Z 994.543,A -85,B 0,C 180,E1 13251.768,E2 13251.768} C_VEL
LIN {X 0,Y 289.327,Z 1001.945,A -85,B 0,C 180,E1 13247.087,E2 13247.087} C_VEL
LIN {X 0,Y 288.424,Z 1006.85,A -85,B 0,C 180,E1 13243.027,E2 13243.027} C_VEL
LIN {X 0,Y 288.039,Z 1010.761,A -85,B 0,C 180,E1 13238.589,E2 13238.589} C_VEL
LIN {X 0,Y 287.962,Z 1012.785,A -85,B 0,C 180,E1 13234.785,E2 13234.785} C_VEL
LIN {X 0,Y 287.975,Z 1013.675,A -85,B 0,C 180,E1 13231.199,E2 13231.199} C_VEL
LIN {X 0,Y 287.959,Z 1013.507,A -85,B 0,C 180,E1 13227.219,E2 13227.219} C_VEL
LIN {X 0,Y 287.969,Z 1011.905,A -85,B 0,C 180,E1 13223.221,E2 13223.221} C_VEL
LIN {X 0,Y 288.115,Z 1009.406,A -85,B 0,C 180,E1 13219.609,E2 13219.609} C_VEL
LIN {X 0,Y 288.704,Z 1005.213,A -85,B 0,C 180,E1 13215.362,E2 13215.362} C_VEL
LIN {X 0,Y 289.939,Z 999.339,A -85,B 0,C 180,E1 13211.092,E2 13211.092} C_VEL
LIN {X 0,Y 292.057,Z 992.024,A -85,B 0,C 180,E1 13206.821,E2 13206.821} C_VEL
LIN {X 0,Y 295.221,Z 982.739,A -85,B 0,C 180,E1 13202.54,E2 13202.54} C_VEL
LIN {X 0,Y 299.501,Z 971.767,A -85,B 0,C 180,E1 13198.351,E2 13198.351} C_VEL
LIN {X 0,Y 304.329,Z 960.11,A -85,B 0,C 180,E1 13194.681,E2 13194.681} C_VEL
LIN {X 0,Y 310.583,Z 945.63,A -85,B 0,C 180,E1 13190.881,E2 13190.881} C_VEL
LIN {X 0,Y 316.755,Z 931.411,A -85,B 0,C 180,E1 13187.76,E2 13187.76} C_VEL
LIN {X 0,Y 323.731,Z 914.973,A -85,B 0,C 180,E1 13184.744,E2 13184.744} C_VEL
LIN {X 0,Y 330.777,Z 897.895,A -85,B 0,C 180,E1 13182.112,E2 13182.112} C_VEL
LIN {X 0,Y 337.692,Z 879.801,A -85,B 0,C 180,E1 13179.804,E2 13179.804} C_VEL
LIN {X 0,Y 344.554,Z 860.737,A -85,B 0,C 180,E1 13177.755,E2 13177.755} C_VEL
LIN {X 0,Y 350.962,Z 840.846,A -85,B 0,C 180,E1 13176.003,E2 13176.003} C_VEL
LIN {X 0,Y 357.271,Z 819.016,A -85,B 0,C 180,E1 13174.424,E2 13174.424} C_VEL
LIN {X 0,Y 362.43,Z 798.31,A -85,B 0,C 180,E1 13173.226,E2 13173.226} C_VEL
LIN {X 0,Y 367.386,Z 774.415,A -85,B 0,C 180,E1 13172.143,E2 13172.143} C_VEL
LIN {X 0,Y 371.274,Z 751.183,A -85,B 0,C 180,E1 13171.358,E2 13171.358} C_VEL
LIN {X 0,Y 373.855,Z 727.553,A -85,B 0,C 180,E1 13170.774,E2 13170.774} C_VEL
LIN {X 0,Y 388.751,Z 518.293,A -85,B 0,C 180,E1 13166.528,E2 13166.528} C_VEL
LIN {X 0,Y 388.948,Z 515.13,A -85,B 0,C 180,E1 13166.454,E2 13166.454} C_VEL
LIN {X 0,Y 378.915,Z 498.841,A -85,B 0,C 180,E1 13163.028,E2 13163.028} C_VEL
LIN {X 0,Y 370.183,Z 485.779,A -85,B 0,C 180,E1 13159.649,E2 13159.649} C_VEL
LIN {X 0,Y 363.716,Z 477.117,A -85,B 0,C 180,E1 13156.859,E2 13156.859} C_VEL
LIN {X 0,Y 359.119,Z 471.324,A -85,B 0,C 180,E1 13154.676,E2 13154.676} C_VEL
LIN {X 0,Y 355.306,Z 466.406,A -85,B 0,C 180,E1 13152.679,E2 13152.679} C_VEL
LIN {X 0,Y 351.501,Z 461.554,A -85,B 0,C 180,E1 13150.489,E2 13150.489} C_VEL
LIN {X 0,Y 347.245,Z 456.562,A -85,B 0,C 180,E1 13147.777,E2 13147.777} C_VEL
LIN {X 0,Y 346.082,Z 455.07,A -85,B 0,C 180,E1 13146.969,E2 13146.969} C_VEL
LIN {X 0,Y 342.605,Z 451.303,A -85,B 0,C 180,E1 13144.351,E2 13144.351} C_VEL
LIN {X 0,Y 341.314,Z 449.176,A -85,B 0,C 180,E1 13143.19,E2 13143.19} C_VEL
LIN {X 0,Y 338.046,Z 446.303,A -85,B 0,C 180,E1 13140.169,E2 13140.169} C_VEL
LIN {X 0,Y 336.148,Z 442.946,A -85,B 0,C 180,E1 13137.862,E2 13137.862} C_VEL
LIN {X 0,Y 332.61,Z 440.279,A -85,B 0,C 180,E1 13132.702,E2 13132.702} C_VEL
LIN {X 0,Y 331.014,Z 437.064,A -85,B 0,C 180,E1 13127.97,E2 13127.97} C_VEL
LIN {X 0,Y 330.494,Z 436.521,A -85,B 0,C 180,E1 13123.116,E2 13123.116} C_VEL
LIN {X 0,Y 331.137,Z 437.203,A -85,B 0,C 180,E1 13118.756,E2 13118.756} C_VEL
LIN {X 0,Y 333.758,Z 441.493,A -85,B 0,C 180,E1 13112.453,E2 13112.453} C_VEL
LIN {X 0,Y 336.447,Z 443.296,A -85,B 0,C 180,E1 13108.961,E2 13108.961} C_VEL
LIN {X 0,Y 338.746,Z 447.155,A -85,B 0,C 180,E1 13106.295,E2 13106.295} C_VEL
LIN {X 0,Y 341.713,Z 449.703,A -85,B 0,C 180,E1 13103.664,E2 13103.664} C_VEL
LIN {X 0,Y 344.846,Z 454.015,A -85,B 0,C 180,E1 13101.117,E2 13101.117} C_VEL
LIN {X 0,Y 346.874,Z 455.899,A -85,B 0,C 180,E1 13099.729,E2 13099.729} C_VEL
LIN {X 0,Y 350.478,Z 460.517,A -85,B 0,C 180,E1 13097.358,E2 13097.358} C_VEL
LIN {X 0,Y 351.905,Z 462.191,A -85,B 0,C 180,E1 13096.498,E2 13096.498} C_VEL
LIN {X 0,Y 356.673,Z 468.126,A -85,B 0,C 180,E1 13093.847,E2 13093.847} C_VEL
LIN {X 0,Y 361.31,Z 474.077,A -85,B 0,C 180,E1 13091.534,E2 13091.534} C_VEL
LIN {X 0,Y 365.86,Z 480.006,A -85,B 0,C 180,E1 13089.462,E2 13089.462} C_VEL
LIN {X 0,Y 372.538,Z 488.778,A -85,B 0,C 180,E1 13086.717,E2 13086.717} C_VEL
LIN {X 0,Y 382.243,Z 502.465,A -85,B 0,C 180,E1 13083.17,E2 13083.17} C_VEL
LIN {X 0,Y 388.569,Z 512.186,A -85,B 0,C 180,E1 13081.077,E2 13081.077} C_VEL
LIN {X 0,Y 373.972,Z 715.604,A -85,B 0,C 180,E1 13076.948,E2 13076.948} C_VEL
LIN {X 0,Y 370.948,Z 740.249,A -85,B 0,C 180,E1 13076.268,E2 13076.268} C_VEL
LIN {X 0,Y 367.256,Z 762.623,A -85,B 0,C 180,E1 13075.424,E2 13075.424} C_VEL
LIN {X 0,Y 362.621,Z 784.443,A -85,B 0,C 180,E1 13074.339,E2 13074.339} C_VEL
LIN {X 0,Y 357.436,Z 805.349,A -85,B 0,C 180,E1 13073.05,E2 13073.05} C_VEL
LIN {X 0,Y 351.565,Z 825.428,A -85,B 0,C 180,E1 13071.518,E2 13071.518} C_VEL
LIN {X 0,Y 344.932,Z 845.772,A -85,B 0,C 180,E1 13069.643,E2 13069.643} C_VEL
LIN {X 0,Y 338.475,Z 863.627,A -85,B 0,C 180,E1 13067.654,E2 13067.654} C_VEL
LIN {X 0,Y 330.88,Z 883.035,A -85,B 0,C 180,E1 13065.057,E2 13065.057} C_VEL
LIN {X 0,Y 324.146,Z 899.189,A -85,B 0,C 180,E1 13062.464,E2 13062.464} C_VEL
LIN {X 0,Y 317.199,Z 914.94,A -85,B 0,C 180,E1 13059.429,E2 13059.429} C_VEL
LIN {X 0,Y 310.712,Z 929.516,A -85,B 0,C 180,E1 13056.089,E2 13056.089} C_VEL
LIN {X 0,Y 305.045,Z 941.994,A -85,B 0,C 180,E1 13052.625,E2 13052.625} C_VEL
LIN {X 0,Y 299.816,Z 953.957,A -85,B 0,C 180,E1 13048.657,E2 13048.657} C_VEL
LIN {X 0,Y 295.798,Z 963.597,A -85,B 0,C 180,E1 13044.759,E2 13044.759} C_VEL
LIN {X 0,Y 292.311,Z 972.942,A -85,B 0,C 180,E1 13040.104,E2 13040.104} C_VEL
LIN {X 0,Y 290.263,Z 979.438,A -85,B 0,C 180,E1 13036.042,E2 13036.042} C_VEL
LIN {X 0,Y 289.354,Z 982.949,A -85,B 0,C 180,E1 13033.335,E2 13033.335} C_VEL
LIN {X 0,Y 287.99,Z 984.777,A -85,B 0,C 180,E1 13031.862,E2 13031.862} C_VEL
LIN {X 0,Y 282.471,Z 988.015,A -85,B 0,C 180,E1 13028.857,E2 13028.857} C_VEL
LIN {X 0,Y 280.323,Z 989.429,A -85,B 0,C 180,E1 13026.992,E2 13026.992} C_VEL
LIN {X 0,Y 280.198,Z 989.693,A -85,B 0,C 180,E1 13026.539,E2 13026.539} C_VEL
LIN {X 0,Y 280.008,Z 991.591,A -85,B 0,C 180,E1 13022.567,E2 13022.567} C_VEL
LIN {X 0,Y 279.992,Z 992.388,A -85,B 0,C 180,E1 13018.988,E2 13018.988} C_VEL
LIN {X 0,Y 280.013,Z 992.203,A -85,B 0,C 180,E1 13014.652,E2 13014.652} C_VEL
LIN {X 0,Y 280.167,Z 990.552,A -85,B 0,C 180,E1 13010.291,E2 13010.291} C_VEL
LIN {X 0,Y 280.644,Z 987.74,A -85,B 0,C 180,E1 13005.989,E2 13005.989} C_VEL
LIN {X 0,Y 281.764,Z 983.295,A -85,B 0,C 180,E1 13001.512,E2 13001.512} C_VEL
LIN {X 0,Y 283.724,Z 977.483,A -85,B 0,C 180,E1 12997.058,E2 12997.058} C_VEL
LIN {X 0,Y 286.854,Z 969.666,A -85,B 0,C 180,E1 12992.466,E2 12992.466} C_VEL
LIN {X 0,Y 291.14,Z 960.428,A -85,B 0,C 180,E1 12988.067,E2 12988.067} C_VEL
LIN {X 0,Y 296.542,Z 949.417,A -85,B 0,C 180,E1 12983.867,E2 12983.867} C_VEL
LIN {X 0,Y 303.357,Z 936.105,A -85,B 0,C 180,E1 12979.708,E2 12979.708} C_VEL
LIN {X 0,Y 310.347,Z 922.645,A -85,B 0,C 180,E1 12976.234,E2 12976.234} C_VEL
LIN {X 0,Y 318.082,Z 907.231,A -85,B 0,C 180,E1 12972.966,E2 12972.966} C_VEL
LIN {X 0,Y 326.108,Z 890.806,A -85,B 0,C 180,E1 12970.065,E2 12970.065} C_VEL
LIN {X 0,Y 333.637,Z 874.38,A -85,B 0,C 180,E1 12967.656,E2 12967.656} C_VEL
LIN {X 0,Y 341.925,Z 854.972,A -85,B 0,C 180,E1 12965.286,E2 12965.286} C_VEL
LIN {X 0,Y 349.01,Z 836.789,A -85,B 0,C 180,E1 12963.45,E2 12963.45} C_VEL
LIN {X 0,Y 356.366,Z 815.683,A -85,B 0,C 180,E1 12961.697,E2 12961.697} C_VEL
LIN {X 0,Y 362.63,Z 795.302,A -85,B 0,C 180,E1 12960.316,E2 12960.316} C_VEL
LIN {X 0,Y 368.231,Z 773.627,A -85,B 0,C 180,E1 12959.145,E2 12959.145} C_VEL
LIN {X 0,Y 373.079,Z 751.017,A -85,B 0,C 180,E1 12958.187,E2 12958.187} C_VEL
LIN {X 0,Y 376.747,Z 728.497,A -85,B 0,C 180,E1 12957.481,E2 12957.481} C_VEL
LIN {X 0,Y 380.118,Z 697.395,A -85,B 0,C 180,E1 12956.77,E2 12956.77} C_VEL
LIN {X 0,Y 397.267,Z 521.73,A -85,B 0,C 180,E1 12953.089,E2 12953.089} C_VEL
LIN {X 0,Y 394.611,Z 516.274,A -85,B 0,C 180,E1 12951.109,E2 12951.109} C_VEL
LIN {X 0,Y 393.201,Z 513.379,A -85,B 0,C 180,E1 12949.776,E2 12949.776} C_VEL
LIN {X 0,Y 392.049,Z 510.774,A -85,B 0,C 180,E1 12948.34,E2 12948.34} C_VEL
LIN {X 0,Y 390.801,Z 507.069,A -85,B 0,C 180,E1 12945.101,E2 12945.101} C_VEL
LIN {X 0,Y 390.811,Z 507.056,A -85,B 0,C 180,E1 12943.349,E2 12943.349} C_VEL
LIN {X 0,Y 391.98,Z 510.701,A -85,B 0,C 180,E1 12940.169,E2 12940.169} C_VEL
LIN {X 0,Y 393.953,Z 514.724,A -85,B 0,C 180,E1 12937.938,E2 12937.938} C_VEL
LIN {X 0,Y 396.189,Z 520.399,A -85,B 0,C 180,E1 12936.027,E2 12936.027} C_VEL
LIN {X 0,Y 397.22,Z 523.33,A -85,B 0,C 180,E1 12935.265,E2 12935.265} C_VEL
LIN {X 0,Y 379.701,Z 703.762,A -85,B 0,C 180,E1 12931.479,E2 12931.479} C_VEL
LIN {X 0,Y 376.235,Z 736.798,A -85,B 0,C 180,E1 12930.739,E2 12930.739} C_VEL
LIN {X 0,Y 372.44,Z 759.664,A -85,B 0,C 180,E1 12930.082,E2 12930.082} C_VEL
LIN {X 0,Y 367.495,Z 782.374,A -85,B 0,C 180,E1 12929.217,E2 12929.217} C_VEL
LIN {X 0,Y 361.917,Z 803.892,A -85,B 0,C 180,E1 12928.152,E2 12928.152} C_VEL
LIN {X 0,Y 355.421,Z 825.084,A -85,B 0,C 180,E1 12926.821,E2 12926.821} C_VEL
LIN {X 0,Y 348.267,Z 846.053,A -85,B 0,C 180,E1 12925.199,E2 12925.199} C_VEL
LIN {X 0,Y 340.839,Z 865.401,A -85,B 0,C 180,E1 12923.357,E2 12923.357} C_VEL
LIN {X 0,Y 332.701,Z 885.124,A -85,B 0,C 180,E1 12921.09,E2 12921.09} C_VEL
LIN {X 0,Y 325.203,Z 902.037,A -85,B 0,C 180,E1 12918.745,E2 12918.745} C_VEL
LIN {X 0,Y 316.633,Z 920.517,A -85,B 0,C 180,E1 12915.667,E2 12915.667} C_VEL
LIN {X 0,Y 309.138,Z 936.323,A -85,B 0,C 180,E1 12912.488,E2 12912.488} C_VEL
LIN {X 0,Y 302.068,Z 950.94,A -85,B 0,C 180,E1 12908.936,E2 12908.936} C_VEL
LIN {X 0,Y 295.844,Z 964.283,A -85,B 0,C 180,E1 12905.073,E2 12905.073} C_VEL
LIN {X 0,Y 290.702,Z 975.659,A -85,B 0,C 180,E1 12901.064,E2 12901.064} C_VEL
LIN {X 0,Y 286.368,Z 986.298,A -85,B 0,C 180,E1 12896.551,E2 12896.551} C_VEL
LIN {X 0,Y 283.541,Z 994.267,A -85,B 0,C 180,E1 12892.391,E2 12892.391} C_VEL
LIN {X 0,Y 281.466,Z 1001.654,A -85,B 0,C 180,E1 12887.58,E2 12887.58} C_VEL
LIN {X 0,Y 280.46,Z 1006.686,A -85,B 0,C 180,E1 12883.283,E2 12883.283} C_VEL
LIN {X 0,Y 280.041,Z 1010.587,A -85,B 0,C 180,E1 12878.63,E2 12878.63} C_VEL
LIN {X 0,Y 279.966,Z 1012.563,A -85,B 0,C 180,E1 12874.717,E2 12874.717} C_VEL
LIN {X 0,Y 279.975,Z 1013.403,A -85,B 0,C 180,E1 12871.028,E2 12871.028} C_VEL
LIN {X 0,Y 279.957,Z 1013.145,A -85,B 0,C 180,E1 12866.935,E2 12866.935} C_VEL
LIN {X 0,Y 279.97,Z 1011.475,A -85,B 0,C 180,E1 12862.825,E2 12862.825} C_VEL
LIN {X 0,Y 280.164,Z 1008.918,A -85,B 0,C 180,E1 12859.103,E2 12859.103} C_VEL
LIN {X 0,Y 280.874,Z 1004.341,A -85,B 0,C 180,E1 12854.521,E2 12854.521} C_VEL
LIN {X 0,Y 282.228,Z 998.656,A -85,B 0,C 180,E1 12850.339,E2 12850.339} C_VEL
LIN {X 0,Y 284.691,Z 990.794,A -85,B 0,C 180,E1 12845.744,E2 12845.744} C_VEL
LIN {X 0,Y 287.97,Z 981.93,A -85,B 0,C 180,E1 12841.604,E2 12841.604} C_VEL
LIN {X 0,Y 292.822,Z 970.227,A -85,B 0,C 180,E1 12837.125,E2 12837.125} C_VEL
LIN {X 0,Y 298.104,Z 958.277,A -85,B 0,C 180,E1 12833.351,E2 12833.351} C_VEL
LIN {X 0,Y 304.435,Z 944.276,A -85,B 0,C 180,E1 12829.692,E2 12829.692} C_VEL
LIN {X 0,Y 311.391,Z 929.025,A -85,B 0,C 180,E1 12826.351,E2 12826.351} C_VEL
LIN {X 0,Y 318.487,Z 912.852,A -85,B 0,C 180,E1 12823.434,E2 12823.434} C_VEL
LIN {X 0,Y 326.214,Z 894.547,A -85,B 0,C 180,E1 12820.669,E2 12820.669} C_VEL
LIN {X 0,Y 333.188,Z 876.865,A -85,B 0,C 180,E1 12818.452,E2 12818.452} C_VEL
LIN {X 0,Y 340.599,Z 856.451,A -85,B 0,C 180,E1 12816.335,E2 12816.335} C_VEL
LIN {X 0,Y 347.333,Z 836.015,A -85,B 0,C 180,E1 12814.594,E2 12814.594} C_VEL
LIN {X 0,Y 353.403,Z 814.799,A -85,B 0,C 180,E1 12813.139,E2 12813.139} C_VEL
LIN {X 0,Y 358.934,Z 792.676,A -85,B 0,C 180,E1 12811.917,E2 12811.917} C_VEL
LIN {X 0,Y 363.379,Z 770.864,A -85,B 0,C 180,E1 12810.985,E2 12810.985} C_VEL
LIN {X 0,Y 367.399,Z 745.78,A -85,B 0,C 180,E1 12810.193,E2 12810.193} C_VEL
LIN {X 0,Y 369.845,Z 722.26,A -85,B 0,C 180,E1 12809.63,E2 12809.63} C_VEL
LIN {X 0,Y 384.663,Z 519.596,A -85,B 0,C 180,E1 12805.519,E2 12805.519} C_VEL
LIN {X 0,Y 375.779,Z 504.962,A -85,B 0,C 180,E1 12802.363,E2 12802.363} C_VEL
LIN {X 0,Y 367.669,Z 492.63,A -85,B 0,C 180,E1 12799.128,E2 12799.128} C_VEL
LIN {X 0,Y 361.47,Z 484.245,A -85,B 0,C 180,E1 12796.387,E2 12796.387} C_VEL
LIN {X 0,Y 356.939,Z 478.463,A -85,B 0,C 180,E1 12794.187,E2 12794.187} C_VEL
LIN {X 0,Y 353.319,Z 473.76,A -85,B 0,C 180,E1 12792.253,E2 12792.253} C_VEL
LIN {X 0,Y 348.908,Z 468.261,A -85,B 0,C 180,E1 12789.65,E2 12789.65} C_VEL
LIN {X 0,Y 345.188,Z 463.471,A -85,B 0,C 180,E1 12787.154,E2 12787.154} C_VEL
LIN {X 0,Y 340.974,Z 458.773,A -85,B 0,C 180,E1 12783.951,E2 12783.951} C_VEL
LIN {X 0,Y 339.802,Z 456.902,A -85,B 0,C 180,E1 12782.867,E2 12782.867} C_VEL
LIN {X 0,Y 336.593,Z 453.928,A -85,B 0,C 180,E1 12779.829,E2 12779.829} C_VEL
LIN {X 0,Y 334.813,Z 450.774,A -85,B 0,C 180,E1 12777.603,E2 12777.603} C_VEL
LIN {X 0,Y 331.338,Z 448.019,A -85,B 0,C 180,E1 12772.369,E2 12772.369} C_VEL
LIN {X 0,Y 329.847,Z 444.938,A -85,B 0,C 180,E1 12767.749,E2 12767.749} C_VEL
LIN {X 0,Y 329.395,Z 444.43,A -85,B 0,C 180,E1 12762.694,E2 12762.694} C_VEL
LIN {X 0,Y 330.089,Z 445.341,A -85,B 0,C 180,E1 12758.499,E2 12758.499} C_VEL
LIN {X 0,Y 332.656,Z 449.462,A -85,B 0,C 180,E1 12752.427,E2 12752.427} C_VEL
LIN {X 0,Y 335.169,Z 451.208,A -85,B 0,C 180,E1 12749.129,E2 12749.129} C_VEL
LIN {X 0,Y 337.541,Z 455.096,A -85,B 0,C 180,E1 12746.362,E2 12746.362} C_VEL
LIN {X 0,Y 340.236,Z 457.42,A -85,B 0,C 180,E1 12743.944,E2 12743.944} C_VEL
LIN {X 0,Y 343.505,Z 461.875,A -85,B 0,C 180,E1 12741.258,E2 12741.258} C_VEL
LIN {X 0,Y 345.308,Z 463.635,A -85,B 0,C 180,E1 12739.997,E2 12739.997} C_VEL
LIN {X 0,Y 348.964,Z 468.275,A -85,B 0,C 180,E1 12737.564,E2 12737.564} C_VEL
LIN {X 0,Y 351.056,Z 471.069,A -85,B 0,C 180,E1 12736.284,E2 12736.284} C_VEL
LIN {X 0,Y 354.762,Z 475.536,A -85,B 0,C 180,E1 12734.227,E2 12734.227} C_VEL
LIN {X 0,Y 359.346,Z 481.52,A -85,B 0,C 180,E1 12731.889,E2 12731.889} C_VEL
LIN {X 0,Y 363.915,Z 487.563,A -85,B 0,C 180,E1 12729.768,E2 12729.768} C_VEL
LIN {X 0,Y 370.444,Z 496.307,A -85,B 0,C 180,E1 12727.036,E2 12727.036} C_VEL
LIN {X 0,Y 379.542,Z 509.299,A -85,B 0,C 180,E1 12723.646,E2 12723.646} C_VEL
LIN {X 0,Y 384.275,Z 516.796,A -85,B 0,C 180,E1 12722.021,E2 12722.021} C_VEL
LIN {X 0,Y 369.493,Z 715.95,A -85,B 0,C 180,E1 12717.968,E2 12717.968} C_VEL
LIN {X 0,Y 366.388,Z 740.537,A -85,B 0,C 180,E1 12717.29,E2 12717.29} C_VEL
LIN {X 0,Y 362.567,Z 763.024,A -85,B 0,C 180,E1 12716.441,E2 12716.441} C_VEL
LIN {X 0,Y 357.632,Z 785.505,A -85,B 0,C 180,E1 12715.319,E2 12715.319} C_VEL
LIN {X 0,Y 352.008,Z 807.251,A -85,B 0,C 180,E1 12713.96,E2 12713.96} C_VEL
LIN {X 0,Y 345.984,Z 827.21,A -85,B 0,C 180,E1 12712.419,E2 12712.419} C_VEL
LIN {X 0,Y 338.966,Z 847.823,A -85,B 0,C 180,E1 12710.481,E2 12710.481} C_VEL
LIN {X 0,Y 331.923,Z 866.604,A -85,B 0,C 180,E1 12708.343,E2 12708.343} C_VEL
LIN {X 0,Y 324.637,Z 884.315,A -85,B 0,C 180,E1 12705.904,E2 12705.904} C_VEL
LIN {X 0,Y 317.258,Z 901.352,A -85,B 0,C 180,E1 12703.11,E2 12703.11} C_VEL
LIN {X 0,Y 310.096,Z 916.878,A -85,B 0,C 180,E1 12700.022,E2 12700.022} C_VEL
LIN {X 0,Y 302.775,Z 932.449,A -85,B 0,C 180,E1 12696.276,E2 12696.276} C_VEL
LIN {X 0,Y 296.984,Z 944.789,A -85,B 0,C 180,E1 12692.696,E2 12692.696} C_VEL
LIN {X 0,Y 291.667,Z 956.32,A -85,B 0,C 180,E1 12688.62,E2 12688.62} C_VEL
LIN {X 0,Y 287.455,Z 966.182,A -85,B 0,C 180,E1 12684.406,E2 12684.406} C_VEL
LIN {X 0,Y 284.254,Z 974.325,A -85,B 0,C 180,E1 12680.032,E2 12680.032} C_VEL
LIN {X 0,Y 282.027,Z 981.198,A -85,B 0,C 180,E1 12675.416,E2 12675.416} C_VEL
LIN {X 0,Y 280.852,Z 985.86,A -85,B 0,C 180,E1 12671.261,E2 12671.261} C_VEL
LIN {X 0,Y 280.223,Z 989.5,A -85,B 0,C 180,E1 12666.886,E2 12666.886} C_VEL
LIN {X 0,Y 280.198,Z 989.693,A -85,B 0,C 180,E1 12666.539,E2 12666.539} C_VEL
LIN {X 0,Y 279.106,Z 990.606,A -85,B 0,C 180,E1 12664.975,E2 12664.975} C_VEL
LIN {X 0,Y 275.074,Z 991.855,A -85,B 0,C 180,E1 12662.455,E2 12662.455} C_VEL
LIN {X 0,Y 272.319,Z 992.521,A -85,B 0,C 180,E1 12660.298,E2 12660.298} C_VEL
LIN {X 0,Y 271.989,Z 992.643,A -85,B 0,C 180,E1 12659.358,E2 12659.358} C_VEL
LIN {X 0,Y 271.997,Z 992.62,A -85,B 0,C 180,E1 12655.43,E2 12655.43} C_VEL
LIN {X 0,Y 272.142,Z 991.252,A -85,B 0,C 180,E1 12650.802,E2 12650.802} C_VEL
LIN {X 0,Y 272.567,Z 988.75,A -85,B 0,C 180,E1 12646.58,E2 12646.58} C_VEL
LIN {X 0,Y 273.734,Z 984.392,A -85,B 0,C 180,E1 12641.667,E2 12641.667} C_VEL
LIN {X 0,Y 275.605,Z 979.012,A -85,B 0,C 180,E1 12637.291,E2 12637.291} C_VEL
LIN {X 0,Y 278.885,Z 971.338,A -85,B 0,C 180,E1 12632.411,E2 12632.411} C_VEL
LIN {X 0,Y 282.961,Z 962.893,A -85,B 0,C 180,E1 12628.161,E2 12628.161} C_VEL
LIN {X 0,Y 288.655,Z 951.96,A -85,B 0,C 180,E1 12623.692,E2 12623.692} C_VEL
LIN {X 0,Y 295.364,Z 939.665,A -85,B 0,C 180,E1 12619.581,E2 12619.581} C_VEL
LIN {X 0,Y 302.7,Z 926.099,A -85,B 0,C 180,E1 12615.913,E2 12615.913} C_VEL
LIN {X 0,Y 310.986,Z 910.626,A -85,B 0,C 180,E1 12612.44,E2 12612.44} C_VEL
LIN {X 0,Y 319.01,Z 895.063,A -85,B 0,C 180,E1 12609.563,E2 12609.563} C_VEL
LIN {X 0,Y 327.686,Z 877.19,A -85,B 0,C 180,E1 12606.835,E2 12606.835} C_VEL
LIN {X 0,Y 335.644,Z 859.701,A -85,B 0,C 180,E1 12604.614,E2 12604.614} C_VEL
LIN {X 0,Y 343.589,Z 840.37,A -85,B 0,C 180,E1 12602.594,E2 12602.594} C_VEL
LIN {X 0,Y 351.005,Z 820.534,A -85,B 0,C 180,E1 12600.881,E2 12600.881} C_VEL
LIN {X 0,Y 357.516,Z 800.502,A -85,B 0,C 180,E1 12599.476,E2 12599.476} C_VEL
LIN {X 0,Y 363.727,Z 778.458,A -85,B 0,C 180,E1 12598.224,E2 12598.224} C_VEL
LIN {X 0,Y 368.503,Z 757.908,A -85,B 0,C 180,E1 12597.309,E2 12597.309} C_VEL
LIN {X 0,Y 372.785,Z 734.632,A -85,B 0,C 180,E1 12596.517,E2 12596.517} C_VEL
LIN {X 0,Y 375.702,Z 712.569,A -85,B 0,C 180,E1 12595.962,E2 12595.962} C_VEL
LIN {X 0,Y 394.612,Z 527.244,A -85,B 0,C 180,E1 12592.081,E2 12592.081} C_VEL
LIN {X 0,Y 392.126,Z 521.697,A -85,B 0,C 180,E1 12589.867,E2 12589.867} C_VEL
LIN {X 0,Y 390.8,Z 518.609,A -85,B 0,C 180,E1 12588.19,E2 12588.19} C_VEL
LIN {X 0,Y 389.654,Z 514.81,A -85,B 0,C 180,E1 12584.675,E2 12584.675} C_VEL
LIN {X 0,Y 389.668,Z 515.101,A -85,B 0,C 180,E1 12583.376,E2 12583.376} C_VEL
LIN {X 0,Y 391.1,Z 519.331,A -85,B 0,C 180,E1 12579.811,E2 12579.811} C_VEL
LIN {X 0,Y 392.893,Z 523.473,A -85,B 0,C 180,E1 12577.796,E2 12577.796} C_VEL
LIN {X 0,Y 394.585,Z 528.2,A -85,B 0,C 180,E1 12576.288,E2 12576.288} C_VEL
LIN {X 0,Y 375.833,Z 713.495,A -85,B 0,C 180,E1 12572.405,E2 12572.405} C_VEL
LIN {X 0,Y 372.677,Z 739.524,A -85,B 0,C 180,E1 12571.798,E2 12571.798} C_VEL
LIN {X 0,Y 368.37,Z 763.572,A -85,B 0,C 180,E1 12571.086,E2 12571.086} C_VEL
LIN {X 0,Y 363.551,Z 784.205,A -85,B 0,C 180,E1 12570.277,E2 12570.277} C_VEL
LIN {X 0,Y 357.499,Z 806.208,A -85,B 0,C 180,E1 12569.167,E2 12569.167} C_VEL
LIN {X 0,Y 351.129,Z 826.035,A -85,B 0,C 180,E1 12567.907,E2 12567.907} C_VEL
LIN {X 0,Y 343.317,Z 847.734,A -85,B 0,C 180,E1 12566.203,E2 12566.203} C_VEL
LIN {X 0,Y 336.066,Z 865.837,A -85,B 0,C 180,E1 12564.465,E2 12564.465} C_VEL
LIN {X 0,Y 327.119,Z 886.47,A -85,B 0,C 180,E1 12562.059,E2 12562.059} C_VEL
LIN {X 0,Y 319.06,Z 903.836,A -85,B 0,C 180,E1 12559.602,E2 12559.602} C_VEL
LIN {X 0,Y 310.657,Z 920.978,A -85,B 0,C 180,E1 12556.673,E2 12556.673} C_VEL
LIN {X 0,Y 302.672,Z 937.018,A -85,B 0,C 180,E1 12553.386,E2 12553.386} C_VEL
LIN {X 0,Y 295.248,Z 951.52,A -85,B 0,C 180,E1 12549.761,E2 12549.761} C_VEL
LIN {X 0,Y 288.419,Z 965.261,A -85,B 0,C 180,E1 12545.625,E2 12545.625} C_VEL
LIN {X 0,Y 283.321,Z 975.966,A -85,B 0,C 180,E1 12541.729,E2 12541.729} C_VEL
LIN {X 0,Y 278.57,Z 986.889,A -85,B 0,C 180,E1 12536.893,E2 12536.893} C_VEL
LIN {X 0,Y 275.633,Z 994.737,A -85,B 0,C 180,E1 12532.619,E2 12532.619} C_VEL
LIN {X 0,Y 273.549,Z 1001.641,A -85,B 0,C 180,E1 12527.886,E2 12527.886} C_VEL
LIN {X 0,Y 272.493,Z 1006.576,A -85,B 0,C 180,E1 12523.504,E2 12523.504} C_VEL
LIN {X 0,Y 272.043,Z 1010.436,A -85,B 0,C 180,E1 12518.636,E2 12518.636} C_VEL
LIN {X 0,Y 271.969,Z 1012.267,A -85,B 0,C 180,E1 12514.856,E2 12514.856} C_VEL
LIN {X 0,Y 271.981,Z 1013.105,A -85,B 0,C 180,E1 12511.059,E2 12511.059} C_VEL
LIN {X 0,Y 271.962,Z 1012.833,A -85,B 0,C 180,E1 12506.844,E2 12506.844} C_VEL
LIN {X 0,Y 271.972,Z 1011.271,A -85,B 0,C 180,E1 12502.825,E2 12502.825} C_VEL
LIN {X 0,Y 272.173,Z 1008.75,A -85,B 0,C 180,E1 12498.993,E2 12498.993} C_VEL
LIN {X 0,Y 272.923,Z 1004.247,A -85,B 0,C 180,E1 12494.277,E2 12494.277} C_VEL
LIN {X 0,Y 274.455,Z 998.283,A -85,B 0,C 180,E1 12489.758,E2 12489.758} C_VEL
LIN {X 0,Y 277.107,Z 990.385,A -85,B 0,C 180,E1 12485.036,E2 12485.036} C_VEL
LIN {X 0,Y 280.618,Z 981.486,A -85,B 0,C 180,E1 12480.789,E2 12480.789} C_VEL
LIN {X 0,Y 285.786,Z 969.734,A -85,B 0,C 180,E1 12476.209,E2 12476.209} C_VEL
LIN {X 0,Y 291.393,Z 957.759,A -85,B 0,C 180,E1 12472.363,E2 12472.363} C_VEL
LIN {X 0,Y 298.05,Z 943.674,A -85,B 0,C 180,E1 12468.642,E2 12468.642} C_VEL
LIN {X 0,Y 305.351,Z 928.335,A -85,B 0,C 180,E1 12465.259,E2 12465.259} C_VEL
LIN {X 0,Y 312.6,Z 912.479,A -85,B 0,C 180,E1 12462.375,E2 12462.375} C_VEL
LIN {X 0,Y 320.547,Z 894.33,A -85,B 0,C 180,E1 12459.616,E2 12459.616} C_VEL
LIN {X 0,Y 327.847,Z 876.418,A -85,B 0,C 180,E1 12457.365,E2 12457.365} C_VEL
LIN {X 0,Y 335.46,Z 856.089,A -85,B 0,C 180,E1 12455.258,E2 12455.258} C_VEL
LIN {X 0,Y 342.408,Z 835.65,A -85,B 0,C 180,E1 12453.517,E2 12453.517} C_VEL
LIN {X 0,Y 348.629,Z 814.531,A -85,B 0,C 180,E1 12452.072,E2 12452.072} C_VEL
LIN {X 0,Y 354.346,Z 792.27,A -85,B 0,C 180,E1 12450.847,E2 12450.847} C_VEL
LIN {X 0,Y 358.843,Z 770.752,A -85,B 0,C 180,E1 12449.934,E2 12449.934} C_VEL
LIN {X 0,Y 362.983,Z 745.524,A -85,B 0,C 180,E1 12449.14,E2 12449.14} C_VEL
LIN {X 0,Y 365.51,Z 721.795,A -85,B 0,C 180,E1 12448.573,E2 12448.573} C_VEL
LIN {X 0,Y 380.475,Z 523.927,A -85,B 0,C 180,E1 12444.553,E2 12444.553} C_VEL
LIN {X 0,Y 371.513,Z 509.145,A -85,B 0,C 180,E1 12441.221,E2 12441.221} C_VEL
LIN {X 0,Y 363.463,Z 496.988,A -85,B 0,C 180,E1 12437.862,E2 12437.862} C_VEL
LIN {X 0,Y 355.848,Z 486.82,A -85,B 0,C 180,E1 12434.241,E2 12434.241} C_VEL
LIN {X 0,Y 351.352,Z 481.108,A -85,B 0,C 180,E1 12431.823,E2 12431.823} C_VEL
LIN {X 0,Y 347.269,Z 475.897,A -85,B 0,C 180,E1 12429.362,E2 12429.362} C_VEL
LIN {X 0,Y 343.589,Z 471.128,A -85,B 0,C 180,E1 12426.852,E2 12426.852} C_VEL
LIN {X 0,Y 339.36,Z 466.241,A -85,B 0,C 180,E1 12423.547,E2 12423.547} C_VEL
LIN {X 0,Y 338.238,Z 464.593,A -85,B 0,C 180,E1 12422.51,E2 12422.51} C_VEL
LIN {X 0,Y 335.062,Z 461.433,A -85,B 0,C 180,E1 12419.401,E2 12419.401} C_VEL
LIN {X 0,Y 333.549,Z 458.631,A -85,B 0,C 180,E1 12417.422,E2 12417.422} C_VEL
LIN {X 0,Y 330.13,Z 455.847,A -85,B 0,C 180,E1 12412.166,E2 12412.166} C_VEL
LIN {X 0,Y 328.722,Z 452.855,A -85,B 0,C 180,E1 12407.706,E2 12407.706} C_VEL
LIN {X 0,Y 328.284,Z 452.354,A -85,B 0,C 180,E1 12402.633,E2 12402.633} C_VEL
LIN {X 0,Y 328.942,Z 453.241,A -85,B 0,C 180,E1 12398.607,E2 12398.607} C_VEL
LIN {X 0,Y 331.525,Z 457.401,A -85,B 0,C 180,E1 12392.446,E2 12392.446} C_VEL
LIN {X 0,Y 333.828,Z 458.967,A -85,B 0,C 180,E1 12389.391,E2 12389.391} C_VEL
LIN {X 0,Y 336.154,Z 462.84,A -85,B 0,C 180,E1 12386.614,E2 12386.614} C_VEL
LIN {X 0,Y 338.85,Z 465.294,A -85,B 0,C 180,E1 12384.145,E2 12384.145} C_VEL
LIN {X 0,Y 342.166,Z 469.732,A -85,B 0,C 180,E1 12381.4,E2 12381.4} C_VEL
LIN {X 0,Y 343.745,Z 471.36,A -85,B 0,C 180,E1 12380.268,E2 12380.268} C_VEL
LIN {X 0,Y 347.44,Z 476.019,A -85,B 0,C 180,E1 12377.781,E2 12377.781} C_VEL
LIN {X 0,Y 353.015,Z 483.192,A -85,B 0,C 180,E1 12374.516,E2 12374.516} C_VEL
LIN {X 0,Y 357.528,Z 489.166,A -85,B 0,C 180,E1 12372.174,E2 12372.174} C_VEL
LIN {X 0,Y 363.847,Z 497.478,A -85,B 0,C 180,E1 12369.262,E2 12369.262} C_VEL
LIN {X 0,Y 371.112,Z 507.778,A -85,B 0,C 180,E1 12366.269,E2 12366.269} C_VEL
LIN {X 0,Y 379.282,Z 519.858,A -85,B 0,C 180,E1 12363.267,E2 12363.267} C_VEL
LIN {X 0,Y 380.05,Z 521.457,A -85,B 0,C 180,E1 12362.982,E2 12362.982} C_VEL
LIN {X 0,Y 364.991,Z 717.65,A -85,B 0,C 180,E1 12358.982,E2 12358.982} C_VEL
LIN {X 0,Y 361.832,Z 741.453,A -85,B 0,C 180,E1 12358.316,E2 12358.316} C_VEL
LIN {X 0,Y 357.976,Z 763.511,A -85,B 0,C 180,E1 12357.482,E2 12357.482} C_VEL
LIN {X 0,Y 353.049,Z 785.348,A -85,B 0,C 180,E1 12356.394,E2 12356.394} C_VEL
LIN {X 0,Y 347.251,Z 807.198,A -85,B 0,C 180,E1 12355.035,E2 12355.035} C_VEL
LIN {X 0,Y 341.036,Z 827.206,A -85,B 0,C 180,E1 12353.493,E2 12353.493} C_VEL
LIN {X 0,Y 333.702,Z 848.111,A -85,B 0,C 180,E1 12351.528,E2 12351.528} C_VEL
LIN {X 0,Y 326.515,Z 866.693,A -85,B 0,C 180,E1 12349.409,E2 12349.409} C_VEL
LIN {X 0,Y 318.936,Z 884.533,A -85,B 0,C 180,E1 12346.945,E2 12346.945} C_VEL
LIN {X 0,Y 311.266,Z 901.59,A -85,B 0,C 180,E1 12344.125,E2 12344.125} C_VEL
LIN {X 0,Y 303.797,Z 917.136,A -85,B 0,C 180,E1 12340.999,E2 12340.999} C_VEL
LIN {X 0,Y 296.382,Z 932.271,A -85,B 0,C 180,E1 12337.329,E2 12337.329} C_VEL
LIN {X 0,Y 290.352,Z 944.487,A -85,B 0,C 180,E1 12333.746,E2 12333.746} C_VEL
LIN {X 0,Y 284.698,Z 956.127,A -85,B 0,C 180,E1 12329.592,E2 12329.592} C_VEL
LIN {X 0,Y 280.18,Z 966.082,A -85,B 0,C 180,E1 12325.287,E2 12325.287} C_VEL
LIN {X 0,Y 276.751,Z 974.234,A -85,B 0,C 180,E1 12320.848,E2 12320.848} C_VEL
LIN {X 0,Y 274.379,Z 980.997,A -85,B 0,C 180,E1 12316.293,E2 12316.293} C_VEL
LIN {X 0,Y 272.976,Z 985.914,A -85,B 0,C 180,E1 12311.855,E2 12311.855} C_VEL
LIN {X 0,Y 272.296,Z 989.475,A -85,B 0,C 180,E1 12307.545,E2 12307.545} C_VEL
LIN {X 0,Y 272.031,Z 991.739,A -85,B 0,C 180,E1 12303.117,E2 12303.117} C_VEL
LIN {X 0,Y 271.989,Z 992.643,A -85,B 0,C 180,E1 12299.358,E2 12299.358} C_VEL
LIN {X 0,Y 271.15,Z 992.856,A -85,B 0,C 180,E1 12297.85,E2 12297.85} C_VEL
LIN {X 0,Y 267.479,Z 992.792,A -85,B 0,C 180,E1 12295.349,E2 12295.349} C_VEL
LIN {X 0,Y 264.398,Z 992.383,A -85,B 0,C 180,E1 12292.886,E2 12292.886} C_VEL
LIN {X 0,Y 264.081,Z 992.111,A -85,B 0,C 180,E1 12291.917,E2 12291.917} C_VEL
LIN {X 0,Y 264.5,Z 989.706,A -85,B 0,C 180,E1 12287.117,E2 12287.117} C_VEL
LIN {X 0,Y 265.422,Z 986.223,A -85,B 0,C 180,E1 12282.694,E2 12282.694} C_VEL
LIN {X 0,Y 267.482,Z 980.557,A -85,B 0,C 180,E1 12277.54,E2 12277.54} C_VEL
LIN {X 0,Y 270.466,Z 973.877,A -85,B 0,C 180,E1 12272.918,E2 12272.918} C_VEL
LIN {X 0,Y 274.96,Z 964.996,A -85,B 0,C 180,E1 12268.094,E2 12268.094} C_VEL
LIN {X 0,Y 280.558,Z 954.91,A -85,B 0,C 180,E1 12263.657,E2 12263.657} C_VEL
LIN {X 0,Y 287.186,Z 943.206,A -85,B 0,C 180,E1 12259.526,E2 12259.526} C_VEL
LIN {X 0,Y 295.185,Z 929.386,A -85,B 0,C 180,E1 12255.522,E2 12255.522} C_VEL
LIN {X 0,Y 303.142,Z 915.346,A -85,B 0,C 180,E1 12252.187,E2 12252.187} C_VEL
LIN {X 0,Y 311.912,Z 899.225,A -85,B 0,C 180,E1 12249.038,E2 12249.038} C_VEL
LIN {X 0,Y 320.539,Z 882.697,A -85,B 0,C 180,E1 12246.358,E2 12246.358} C_VEL
LIN {X 0,Y 329.002,Z 865.027,A -85,B 0,C 180,E1 12244.009,E2 12244.009} C_VEL
LIN {X 0,Y 337.167,Z 846.736,A -85,B 0,C 180,E1 12241.978,E2 12241.978} C_VEL
LIN {X 0,Y 344.75,Z 827.65,A -85,B 0,C 180,E1 12240.241,E2 12240.241} C_VEL
LIN {X 0,Y 352.102,Z 807.072,A -85,B 0,C 180,E1 12238.699,E2 12238.699} C_VEL
LIN {X 0,Y 358.088,Z 787.497,A -85,B 0,C 180,E1 12237.512,E2 12237.512} C_VEL
LIN {X 0,Y 364.088,Z 764.452,A -85,B 0,C 180,E1 12236.399,E2 12236.399} C_VEL
LIN {X 0,Y 368.321,Z 744.029,A -85,B 0,C 180,E1 12235.636,E2 12235.636} C_VEL
LIN {X 0,Y 372.167,Z 719.27,A -85,B 0,C 180,E1 12234.958,E2 12234.958} C_VEL
LIN {X 0,Y 392.166,Z 532.749,A -85,B 0,C 180,E1 12231.053,E2 12231.053} C_VEL
LIN {X 0,Y 390.436,Z 528.81,A -85,B 0,C 180,E1 12229.301,E2 12229.301} C_VEL
LIN {X 0,Y 389.418,Z 526.259,A -85,B 0,C 180,E1 12227.846,E2 12227.846} C_VEL
LIN {X 0,Y 388.52,Z 522.706,A -85,B 0,C 180,E1 12224.476,E2 12224.476} C_VEL
LIN {X 0,Y 388.526,Z 523.035,A -85,B 0,C 180,E1 12223.479,E2 12223.479} C_VEL
LIN {X 0,Y 389.763,Z 527.066,A -85,B 0,C 180,E1 12220.051,E2 12220.051} C_VEL
LIN {X 0,Y 391.396,Z 531.06,A -85,B 0,C 180,E1 12218.102,E2 12218.102} C_VEL
LIN {X 0,Y 392.15,Z 533.505,A -85,B 0,C 180,E1 12217.32,E2 12217.32} C_VEL
LIN {X 0,Y 370.982,Z 731.746,A -85,B 0,C 180,E1 12213.154,E2 12213.154} C_VEL
LIN {X 0,Y 366.788,Z 756.159,A -85,B 0,C 180,E1 12212.489,E2 12212.489} C_VEL
LIN {X 0,Y 361.364,Z 780.019,A -85,B 0,C 180,E1 12211.632,E2 12211.632} C_VEL
LIN {X 0,Y 355.279,Z 801.968,A -85,B 0,C 180,E1 12210.583,E2 12210.583} C_VEL
LIN {X 0,Y 348.213,Z 823.605,A -85,B 0,C 180,E1 12209.263,E2 12209.263} C_VEL
LIN {X 0,Y 340.34,Z 845.026,A -85,B 0,C 180,E1 12207.637,E2 12207.637} C_VEL
LIN {X 0,Y 332.016,Z 865,A -85,B 0,C 180,E1 12205.746,E2 12205.746} C_VEL
LIN {X 0,Y 322.744,Z 885.574,A -85,B 0,C 180,E1 12203.363,E2 12203.363} C_VEL
LIN {X 0,Y 314.07,Z 903.486,A -85,B 0,C 180,E1 12200.828,E2 12200.828} C_VEL
LIN {X 0,Y 304.925,Z 921.247,A -85,B 0,C 180,E1 12197.764,E2 12197.764} C_VEL
LIN {X 0,Y 296.704,Z 936.9,A -85,B 0,C 180,E1 12194.507,E2 12194.507} C_VEL
LIN {X 0,Y 288.934,Z 951.298,A -85,B 0,C 180,E1 12190.852,E2 12190.852} C_VEL
LIN {X 0,Y 281.649,Z 965.092,A -85,B 0,C 180,E1 12186.618,E2 12186.618} C_VEL
LIN {X 0,Y 275.964,Z 976.331,A -85,B 0,C 180,E1 12182.416,E2 12182.416} C_VEL
LIN {X 0,Y 271.15,Z 986.648,A -85,B 0,C 180,E1 12177.691,E2 12177.691} C_VEL
LIN {X 0,Y 267.854,Z 994.856,A -85,B 0,C 180,E1 12173.081,E2 12173.081} C_VEL
LIN {X 0,Y 265.638,Z 1001.634,A -85,B 0,C 180,E1 12168.21,E2 12168.21} C_VEL
LIN {X 0,Y 264.497,Z 1006.653,A -85,B 0,C 180,E1 12163.56,E2 12163.56} C_VEL
LIN {X 0,Y 264.046,Z 1010.249,A -85,B 0,C 180,E1 12158.717,E2 12158.717} C_VEL
LIN {X 0,Y 263.973,Z 1012.049,A -85,B 0,C 180,E1 12154.786,E2 12154.786} C_VEL
LIN {X 0,Y 263.984,Z 1012.887,A -85,B 0,C 180,E1 12150.44,E2 12150.44} C_VEL
LIN {X 0,Y 263.974,Z 1012.316,A -85,B 0,C 180,E1 12146.096,E2 12146.096} C_VEL
LIN {X 0,Y 264.002,Z 1010.717,A -85,B 0,C 180,E1 12142.17,E2 12142.17} C_VEL
LIN {X 0,Y 264.295,Z 1007.754,A -85,B 0,C 180,E1 12137.775,E2 12137.775} C_VEL
LIN {X 0,Y 265.293,Z 1002.83,A -85,B 0,C 180,E1 12132.911,E2 12132.911} C_VEL
LIN {X 0,Y 267.198,Z 996.448,A -85,B 0,C 180,E1 12128.126,E2 12128.126} C_VEL
LIN {X 0,Y 270.225,Z 988.275,A -85,B 0,C 180,E1 12123.41,E2 12123.41} C_VEL
LIN {X 0,Y 274.453,Z 978.609,A -85,B 0,C 180,E1 12118.855,E2 12118.855} C_VEL
LIN {X 0,Y 279.687,Z 967.439,A -85,B 0,C 180,E1 12114.618,E2 12114.618} C_VEL
LIN {X 0,Y 286.491,Z 953.647,A -85,B 0,C 180,E1 12110.316,E2 12110.316} C_VEL
LIN {X 0,Y 293.4,Z 939.86,A -85,B 0,C 180,E1 12106.775,E2 12106.775} C_VEL
LIN {X 0,Y 300.784,Z 924.756,A -85,B 0,C 180,E1 12103.568,E2 12103.568} C_VEL
LIN {X 0,Y 308.646,Z 908.213,A -85,B 0,C 180,E1 12100.627,E2 12100.627} C_VEL
LIN {X 0,Y 316.653,Z 890.176,A -85,B 0,C 180,E1 12098.004,E2 12098.004} C_VEL
LIN {X 0,Y 324.79,Z 870.616,A -85,B 0,C 180,E1 12095.648,E2 12095.648} C_VEL
LIN {X 0,Y 331.639,Z 852.474,A -85,B 0,C 180,E1 12093.85,E2 12093.85} C_VEL
LIN {X 0,Y 339.166,Z 830.238,A -85,B 0,C 180,E1 12092.048,E2 12092.048} C_VEL
LIN {X 0,Y 344.817,Z 811.204,A -85,B 0,C 180,E1 12090.796,E2 12090.796} C_VEL
LIN {X 0,Y 350.654,Z 788.202,A -85,B 0,C 180,E1 12089.591,E2 12089.591} C_VEL
LIN {X 0,Y 355.086,Z 767.201,A -85,B 0,C 180,E1 12088.736,E2 12088.736} C_VEL
LIN {X 0,Y 358.857,Z 743.732,A -85,B 0,C 180,E1 12088.025,E2 12088.025} C_VEL
LIN {X 0,Y 361.416,Z 719.411,A -85,B 0,C 180,E1 12087.454,E2 12087.454} C_VEL
LIN {X 0,Y 376.333,Z 528.372,A -85,B 0,C 180,E1 12083.566,E2 12083.566} C_VEL
LIN {X 0,Y 368.448,Z 515.286,A -85,B 0,C 180,E1 12080.532,E2 12080.532} C_VEL
LIN {X 0,Y 361.167,Z 504.094,A -85,B 0,C 180,E1 12077.396,E2 12077.396} C_VEL
LIN {X 0,Y 353.821,Z 494.126,A -85,B 0,C 180,E1 12073.814,E2 12073.814} C_VEL
LIN {X 0,Y 349.406,Z 488.449,A -85,B 0,C 180,E1 12071.387,E2 12071.387} C_VEL
LIN {X 0,Y 345.512,Z 483.408,A -85,B 0,C 180,E1 12068.99,E2 12068.99} C_VEL
LIN {X 0,Y 341.336,Z 478.051,A -85,B 0,C 180,E1 12066.053,E2 12066.053} C_VEL
LIN {X 0,Y 337.76,Z 473.708,A -85,B 0,C 180,E1 12063.139,E2 12063.139} C_VEL
LIN {X 0,Y 336.745,Z 472.322,A -85,B 0,C 180,E1 12062.212,E2 12062.212} C_VEL
LIN {X 0,Y 333.616,Z 469.049,A -85,B 0,C 180,E1 12059.055,E2 12059.055} C_VEL
LIN {X 0,Y 332.265,Z 466.485,A -85,B 0,C 180,E1 12057.24,E2 12057.24} C_VEL
LIN {X 0,Y 328.913,Z 463.673,A -85,B 0,C 180,E1 12051.961,E2 12051.961} C_VEL
LIN {X 0,Y 327.56,Z 460.733,A -85,B 0,C 180,E1 12047.483,E2 12047.483} C_VEL
LIN {X 0,Y 327.181,Z 460.287,A -85,B 0,C 180,E1 12042.43,E2 12042.43} C_VEL
LIN {X 0,Y 327.794,Z 461.139,A -85,B 0,C 180,E1 12038.716,E2 12038.716} C_VEL
LIN {X 0,Y 330.306,Z 465.258,A -85,B 0,C 180,E1 12032.605,E2 12032.605} C_VEL
LIN {X 0,Y 332.546,Z 466.863,A -85,B 0,C 180,E1 12029.57,E2 12029.57} C_VEL
LIN {X 0,Y 334.951,Z 470.78,A -85,B 0,C 180,E1 12026.683,E2 12026.683} C_VEL
LIN {X 0,Y 337.429,Z 473.079,A -85,B 0,C 180,E1 12024.39,E2 12024.39} C_VEL
LIN {X 0,Y 340.952,Z 477.699,A -85,B 0,C 180,E1 12021.452,E2 12021.452} C_VEL
LIN {X 0,Y 342.319,Z 479.293,A -85,B 0,C 180,E1 12020.444,E2 12020.444} C_VEL
LIN {X 0,Y 346.839,Z 485.087,A -85,B 0,C 180,E1 12017.411,E2 12017.411} C_VEL
LIN {X 0,Y 351.271,Z 490.842,A -85,B 0,C 180,E1 12014.808,E2 12014.808} C_VEL
LIN {X 0,Y 355.561,Z 496.582,A -85,B 0,C 180,E1 12012.543,E2 12012.543} C_VEL
LIN {X 0,Y 361.754,Z 504.89,A -85,B 0,C 180,E1 12009.628,E2 12009.628} C_VEL
LIN {X 0,Y 368.752,Z 514.952,A -85,B 0,C 180,E1 12006.686,E2 12006.686} C_VEL
LIN {X 0,Y 375.95,Z 525.662,A -85,B 0,C 180,E1 12003.975,E2 12003.975} C_VEL
LIN {X 0,Y 360.798,Z 716.882,A -85,B 0,C 180,E1 12000.071,E2 12000.071} C_VEL
LIN {X 0,Y 357.531,Z 741.264,A -85,B 0,C 180,E1 11999.398,E2 11999.398} C_VEL
LIN {X 0,Y 353.488,Z 763.801,A -85,B 0,C 180,E1 11998.551,E2 11998.551} C_VEL
LIN {X 0,Y 348.581,Z 785.072,A -85,B 0,C 180,E1 11997.498,E2 11997.498} C_VEL
LIN {X 0,Y 342.918,Z 806.124,A -85,B 0,C 180,E1 11996.209,E2 11996.209} C_VEL
LIN {X 0,Y 336.497,Z 826.332,A -85,B 0,C 180,E1 11994.67,E2 11994.67} C_VEL
LIN {X 0,Y 329.204,Z 846.739,A -85,B 0,C 180,E1 11992.78,E2 11992.78} C_VEL
LIN {X 0,Y 321.948,Z 864.938,A -85,B 0,C 180,E1 11990.729,E2 11990.729} C_VEL
LIN {X 0,Y 313.576,Z 884.155,A -85,B 0,C 180,E1 11988.107,E2 11988.107} C_VEL
LIN {X 0,Y 305.818,Z 900.873,A -85,B 0,C 180,E1 11985.351,E2 11985.351} C_VEL
LIN {X 0,Y 298.005,Z 916.571,A -85,B 0,C 180,E1 11982.197,E2 11982.197} C_VEL
LIN {X 0,Y 290.615,Z 931.068,A -85,B 0,C 180,E1 11978.701,E2 11978.701} C_VEL
LIN {X 0,Y 284.034,Z 943.731,A -85,B 0,C 180,E1 11974.979,E2 11974.979} C_VEL
LIN {X 0,Y 277.806,Z 955.937,A -85,B 0,C 180,E1 11970.613,E2 11970.613} C_VEL
LIN {X 0,Y 273.159,Z 965.491,A -85,B 0,C 180,E1 11966.427,E2 11966.427} C_VEL
LIN {X 0,Y 269.263,Z 974.189,A -85,B 0,C 180,E1 11961.668,E2 11961.668} C_VEL
LIN {X 0,Y 266.682,Z 981.023,A -85,B 0,C 180,E1 11956.994,E2 11956.994} C_VEL
LIN {X 0,Y 265.123,Z 986.011,A -85,B 0,C 180,E1 11952.435,E2 11952.435} C_VEL
LIN {X 0,Y 264.363,Z 989.613,A -85,B 0,C 180,E1 11948.005,E2 11948.005} C_VEL
LIN {X 0,Y 264.041,Z 992.043,A -85,B 0,C 180,E1 11943.211,E2 11943.211} C_VEL
LIN {X 0,Y 263.995,Z 992.945,A -85,B 0,C 180,E1 11939.348,E2 11939.348} C_VEL
LIN {X 0,Y 264.009,Z 992.921,A -85,B 0,C 180,E1 11935.269,E2 11935.269} C_VEL
LIN {X 0,Y 264.081,Z 992.111,A -85,B 0,C 180,E1 11931.917,E2 11931.917} C_VEL
LIN {X 0,Y 263.19,Z 991.61,A -85,B 0,C 180,E1 11930.245,E2 11930.245} C_VEL
LIN {X 0,Y 259.073,Z 990.353,A -85,B 0,C 180,E1 11927.187,E2 11927.187} C_VEL
LIN {X 0,Y 257.089,Z 988.967,A -85,B 0,C 180,E1 11925.009,E2 11925.009} C_VEL
LIN {X 0,Y 257.032,Z 988.37,A -85,B 0,C 180,E1 11924.272,E2 11924.272} C_VEL
LIN {X 0,Y 258.617,Z 983.763,A -85,B 0,C 180,E1 11919.348,E2 11919.348} C_VEL
LIN {X 0,Y 261.436,Z 977.536,A -85,B 0,C 180,E1 11914.294,E2 11914.294} C_VEL
LIN {X 0,Y 265.414,Z 969.824,A -85,B 0,C 180,E1 11909.508,E2 11909.508} C_VEL
LIN {X 0,Y 271.395,Z 959.381,A -85,B 0,C 180,E1 11904.37,E2 11904.37} C_VEL
LIN {X 0,Y 278.163,Z 948.233,A -85,B 0,C 180,E1 11899.968,E2 11899.968} C_VEL
LIN {X 0,Y 285.601,Z 935.921,A -85,B 0,C 180,E1 11896.056,E2 11896.056} C_VEL
LIN {X 0,Y 294.148,Z 921.857,A -85,B 0,C 180,E1 11892.366,E2 11892.366} C_VEL
LIN {X 0,Y 303.01,Z 906.642,A -85,B 0,C 180,E1 11889.114,E2 11889.114} C_VEL
LIN {X 0,Y 312.709,Z 889.089,A -85,B 0,C 180,E1 11886.043,E2 11886.043} C_VEL
LIN {X 0,Y 321.703,Z 871.82,A -85,B 0,C 180,E1 11883.564,E2 11883.564} C_VEL
LIN {X 0,Y 330.48,Z 853.267,A -85,B 0,C 180,E1 11881.387,E2 11881.387} C_VEL
LIN {X 0,Y 339.332,Z 832.734,A -85,B 0,C 180,E1 11879.41,E2 11879.41} C_VEL
LIN {X 0,Y 346.482,Z 813.905,A -85,B 0,C 180,E1 11877.933,E2 11877.933} C_VEL
LIN {X 0,Y 353.897,Z 791.668,A -85,B 0,C 180,E1 11876.518,E2 11876.518} C_VEL
LIN {X 0,Y 359.56,Z 771.471,A -85,B 0,C 180,E1 11875.495,E2 11875.495} C_VEL
LIN {X 0,Y 364.889,Z 748.168,A -85,B 0,C 180,E1 11874.578,E2 11874.578} C_VEL
LIN {X 0,Y 368.969,Z 724.945,A -85,B 0,C 180,E1 11873.906,E2 11873.906} C_VEL
LIN {X 0,Y 389.899,Z 538.579,A -85,B 0,C 180,E1 11870.014,E2 11870.014} C_VEL
LIN {X 0,Y 388.264,Z 534.207,A -85,B 0,C 180,E1 11867.81,E2 11867.81} C_VEL
LIN {X 0,Y 387.397,Z 530.623,A -85,B 0,C 180,E1 11864.43,E2 11864.43} C_VEL
LIN {X 0,Y 387.387,Z 530.965,A -85,B 0,C 180,E1 11863.584,E2 11863.584} C_VEL
LIN {X 0,Y 388.455,Z 534.8,A -85,B 0,C 180,E1 11860.295,E2 11860.295} C_VEL
LIN {X 0,Y 389.907,Z 538.65,A -85,B 0,C 180,E1 11858.409,E2 11858.409} C_VEL
LIN {X 0,Y 389.333,Z 543.989,A -85,B 0,C 180,E1 11858.262,E2 11858.262} C_VEL
LIN {X 0,Y 368.469,Z 731.05,A -85,B 0,C 180,E1 11854.349,E2 11854.349} C_VEL
LIN {X 0,Y 364.273,Z 754.935,A -85,B 0,C 180,E1 11853.71,E2 11853.71} C_VEL
LIN {X 0,Y 358.866,Z 778.237,A -85,B 0,C 180,E1 11852.901,E2 11852.901} C_VEL
LIN {X 0,Y 352.593,Z 800.242,A -85,B 0,C 180,E1 11851.879,E2 11851.879} C_VEL
LIN {X 0,Y 345.071,Z 822.628,A -85,B 0,C 180,E1 11850.547,E2 11850.547} C_VEL
LIN {X 0,Y 336.781,Z 844.411,A -85,B 0,C 180,E1 11848.917,E2 11848.917} C_VEL
LIN {X 0,Y 327.905,Z 864.89,A -85,B 0,C 180,E1 11846.991,E2 11846.991} C_VEL
LIN {X 0,Y 318.255,Z 885.372,A -85,B 0,C 180,E1 11844.619,E2 11844.619} C_VEL
LIN {X 0,Y 309.484,Z 902.711,A -85,B 0,C 180,E1 11842.168,E2 11842.168} C_VEL
LIN {X 0,Y 300.068,Z 920.224,A -85,B 0,C 180,E1 11839.152,E2 11839.152} C_VEL
LIN {X 0,Y 291.212,Z 936.239,A -85,B 0,C 180,E1 11835.815,E2 11835.815} C_VEL
LIN {X 0,Y 282.928,Z 950.761,A -85,B 0,C 180,E1 11832.088,E2 11832.088} C_VEL
LIN {X 0,Y 275.299,Z 964.356,A -85,B 0,C 180,E1 11827.869,E2 11827.869} C_VEL
LIN {X 0,Y 269.228,Z 975.586,A -85,B 0,C 180,E1 11823.603,E2 11823.603} C_VEL
LIN {X 0,Y 264.001,Z 986.002,A -85,B 0,C 180,E1 11818.755,E2 11818.755} C_VEL
LIN {X 0,Y 260.525,Z 993.874,A -85,B 0,C 180,E1 11814.251,E2 11814.251} C_VEL
LIN {X 0,Y 257.896,Z 1001.1,A -85,B 0,C 180,E1 11809.011,E2 11809.011} C_VEL
LIN {X 0,Y 256.682,Z 1005.72,A -85,B 0,C 180,E1 11804.672,E2 11804.672} C_VEL
LIN {X 0,Y 256.076,Z 1009.589,A -85,B 0,C 180,E1 11799.671,E2 11799.671} C_VEL
LIN {X 0,Y 255.976,Z 1011.606,A -85,B 0,C 180,E1 11795.385,E2 11795.385} C_VEL
LIN {X 0,Y 255.998,Z 1012.483,A -85,B 0,C 180,E1 11791.349,E2 11791.349} C_VEL
LIN {X 0,Y 255.972,Z 1012.273,A -85,B 0,C 180,E1 11786.871,E2 11786.871} C_VEL
LIN {X 0,Y 255.983,Z 1010.74,A -85,B 0,C 180,E1 11782.6,E2 11782.6} C_VEL
LIN {X 0,Y 256.215,Z 1008.241,A -85,B 0,C 180,E1 11778.527,E2 11778.527} C_VEL
LIN {X 0,Y 257.038,Z 1004.037,A -85,B 0,C 180,E1 11773.742,E2 11773.742} C_VEL
LIN {X 0,Y 258.755,Z 998.137,A -85,B 0,C 180,E1 11768.946,E2 11768.946} C_VEL
LIN {X 0,Y 261.735,Z 990.367,A -85,B 0,C 180,E1 11763.947,E2 11763.947} C_VEL
LIN {X 0,Y 265.868,Z 981.043,A -85,B 0,C 180,E1 11759.247,E2 11759.247} C_VEL
LIN {X 0,Y 271.682,Z 969.219,A -85,B 0,C 180,E1 11754.422,E2 11754.422} C_VEL
LIN {X 0,Y 277.87,Z 957.3,A -85,B 0,C 180,E1 11750.448,E2 11750.448} C_VEL
LIN {X 0,Y 285.187,Z 943.203,A -85,B 0,C 180,E1 11746.603,E2 11746.603} C_VEL
LIN {X 0,Y 293.153,Z 927.838,A -85,B 0,C 180,E1 11743.132,E2 11743.132} C_VEL
LIN {X 0,Y 300.99,Z 911.943,A -85,B 0,C 180,E1 11740.189,E2 11740.189} C_VEL
LIN {X 0,Y 309.568,Z 893.716,A -85,B 0,C 180,E1 11737.387,E2 11737.387} C_VEL
LIN {X 0,Y 317.288,Z 875.998,A -85,B 0,C 180,E1 11735.151,E2 11735.151} C_VEL
LIN {X 0,Y 325.49,Z 855.413,A -85,B 0,C 180,E1 11733.017,E2 11733.017} C_VEL
LIN {X 0,Y 332.83,Z 835.011,A -85,B 0,C 180,E1 11731.289,E2 11731.289} C_VEL
LIN {X 0,Y 339.364,Z 813.974,A -85,B 0,C 180,E1 11729.862,E2 11729.862} C_VEL
LIN {X 0,Y 345.261,Z 792.222,A -85,B 0,C 180,E1 11728.674,E2 11728.674} C_VEL
LIN {X 0,Y 350.03,Z 770.628,A -85,B 0,C 180,E1 11727.765,E2 11727.765} C_VEL
LIN {X 0,Y 354.294,Z 746.15,A -85,B 0,C 180,E1 11726.994,E2 11726.994} C_VEL
LIN {X 0,Y 356.914,Z 723.314,A -85,B 0,C 180,E1 11726.445,E2 11726.445} C_VEL
LIN {X 0,Y 372.269,Z 532.87,A -85,B 0,C 180,E1 11722.565,E2 11722.565} C_VEL
LIN {X 0,Y 365.614,Z 521.71,A -85,B 0,C 180,E1 11719.905,E2 11719.905} C_VEL
LIN {X 0,Y 358.896,Z 511.197,A -85,B 0,C 180,E1 11716.925,E2 11716.925} C_VEL
LIN {X 0,Y 351.801,Z 501.443,A -85,B 0,C 180,E1 11713.393,E2 11713.393} C_VEL
LIN {X 0,Y 347.474,Z 495.783,A -85,B 0,C 180,E1 11710.947,E2 11710.947} C_VEL
LIN {X 0,Y 343.649,Z 490.787,A -85,B 0,C 180,E1 11708.533,E2 11708.533} C_VEL
LIN {X 0,Y 339.772,Z 485.706,A -85,B 0,C 180,E1 11705.742,E2 11705.742} C_VEL
LIN {X 0,Y 336.155,Z 481.17,A -85,B 0,C 180,E1 11702.727,E2 11702.727} C_VEL
LIN {X 0,Y 335.227,Z 480.024,A -85,B 0,C 180,E1 11701.88,E2 11701.88} C_VEL
LIN {X 0,Y 332.18,Z 476.662,A -85,B 0,C 180,E1 11698.706,E2 11698.706} C_VEL
LIN {X 0,Y 330.977,Z 474.336,A -85,B 0,C 180,E1 11697.056,E2 11697.056} C_VEL
LIN {X 0,Y 327.684,Z 471.498,A -85,B 0,C 180,E1 11691.754,E2 11691.754} C_VEL
LIN {X 0,Y 326.43,Z 468.648,A -85,B 0,C 180,E1 11687.439,E2 11687.439} C_VEL
LIN {X 0,Y 326.058,Z 468.206,A -85,B 0,C 180,E1 11682.472,E2 11682.472} C_VEL
LIN {X 0,Y 326.638,Z 469.036,A -85,B 0,C 180,E1 11678.825,E2 11678.825} C_VEL
LIN {X 0,Y 329.128,Z 473.155,A -85,B 0,C 180,E1 11672.695,E2 11672.695} C_VEL
LIN {X 0,Y 331.22,Z 474.629,A -85,B 0,C 180,E1 11669.826,E2 11669.826} C_VEL
LIN {X 0,Y 333.572,Z 478.524,A -85,B 0,C 180,E1 11666.938,E2 11666.938} C_VEL
LIN {X 0,Y 335.979,Z 480.803,A -85,B 0,C 180,E1 11664.665,E2 11664.665} C_VEL
LIN {X 0,Y 339.49,Z 485.441,A -85,B 0,C 180,E1 11661.686,E2 11661.686} C_VEL
LIN {X 0,Y 340.823,Z 487.091,A -85,B 0,C 180,E1 11660.678,E2 11660.678} C_VEL
LIN {X 0,Y 345.16,Z 492.714,A -85,B 0,C 180,E1 11657.717,E2 11657.717} C_VEL
LIN {X 0,Y 349.535,Z 498.487,A -85,B 0,C 180,E1 11655.102,E2 11655.102} C_VEL
LIN {X 0,Y 353.951,Z 504.48,A -85,B 0,C 180,E1 11652.738,E2 11652.738} C_VEL
LIN {X 0,Y 359.836,Z 512.551,A -85,B 0,C 180,E1 11649.922,E2 11649.922} C_VEL
LIN {X 0,Y 366.391,Z 522.11,A -85,B 0,C 180,E1 11647.111,E2 11647.111} C_VEL
LIN {X 0,Y 371.871,Z 530.529,A -85,B 0,C 180,E1 11644.967,E2 11644.967} C_VEL
LIN {X 0,Y 356.519,Z 718.305,A -85,B 0,C 180,E1 11641.136,E2 11641.136} C_VEL
LIN {X 0,Y 353.195,Z 742.045,A -85,B 0,C 180,E1 11640.475,E2 11640.475} C_VEL
LIN {X 0,Y 349.125,Z 764.09,A -85,B 0,C 180,E1 11639.646,E2 11639.646} C_VEL
LIN {X 0,Y 343.925,Z 785.975,A -85,B 0,C 180,E1 11638.564,E2 11638.564} C_VEL
LIN {X 0,Y 337.789,Z 807.871,A -85,B 0,C 180,E1 11637.208,E2 11637.208} C_VEL
LIN {X 0,Y 331.283,Z 827.699,A -85,B 0,C 180,E1 11635.685,E2 11635.685} C_VEL
LIN {X 0,Y 323.404,Z 848.88,A -85,B 0,C 180,E1 11633.692,E2 11633.692} C_VEL
LIN {X 0,Y 315.701,Z 867.584,A -85,B 0,C 180,E1 11631.548,E2 11631.548} C_VEL
LIN {X 0,Y 307.594,Z 885.37,A -85,B 0,C 180,E1 11629.062,E2 11629.062} C_VEL
LIN {X 0,Y 299.572,Z 901.99,A -85,B 0,C 180,E1 11626.276,E2 11626.276} C_VEL
LIN {X 0,Y 291.48,Z 917.602,A -85,B 0,C 180,E1 11623.079,E2 11623.079} C_VEL
LIN {X 0,Y 283.424,Z 932.699,A -85,B 0,C 180,E1 11619.333,E2 11619.333} C_VEL
LIN {X 0,Y 276.736,Z 945.056,A -85,B 0,C 180,E1 11615.593,E2 11615.593} C_VEL
LIN {X 0,Y 270.452,Z 956.729,A -85,B 0,C 180,E1 11611.265,E2 11611.265} C_VEL
LIN {X 0,Y 265.386,Z 966.703,A -85,B 0,C 180,E1 11606.755,E2 11606.755} C_VEL
LIN {X 0,Y 261.482,Z 974.918,A -85,B 0,C 180,E1 11602.045,E2 11602.045} C_VEL
LIN {X 0,Y 258.693,Z 981.874,A -85,B 0,C 180,E1 11597.04,E2 11597.04} C_VEL
LIN {X 0,Y 257.165,Z 986.529,A -85,B 0,C 180,E1 11592.574,E2 11592.574} C_VEL
LIN {X 0,Y 256.371,Z 990.086,A -85,B 0,C 180,E1 11588.007,E2 11588.007} C_VEL
LIN {X 0,Y 256.05,Z 992.343,A -85,B 0,C 180,E1 11583.311,E2 11583.311} C_VEL
LIN {X 0,Y 255.997,Z 993.229,A -85,B 0,C 180,E1 11579.481,E2 11579.481} C_VEL
LIN {X 0,Y 256.007,Z 993.255,A -85,B 0,C 180,E1 11575.496,E2 11575.496} C_VEL
LIN {X 0,Y 256.175,Z 992.039,A -85,B 0,C 180,E1 11570.607,E2 11570.607} C_VEL
LIN {X 0,Y 256.674,Z 989.601,A -85,B 0,C 180,E1 11566.095,E2 11566.095} C_VEL
LIN {X 0,Y 257.032,Z 988.37,A -85,B 0,C 180,E1 11564.272,E2 11564.272} C_VEL
LIN {X 0,Y 256.466,Z 987.003,A -85,B 0,C 180,E1 11562.572,E2 11562.572} C_VEL
LIN {X 0,Y 251.989,Z 983.175,A -85,B 0,C 180,E1 11557.829,E2 11557.829} C_VEL
LIN {X 0,Y 252.048,Z 981.677,A -85,B 0,C 180,E1 11556.478,E2 11556.478} C_VEL
LIN {X 0,Y 255.404,Z 975.175,A -85,B 0,C 180,E1 11551.641,E2 11551.641} C_VEL
LIN {X 0,Y 260.632,Z 966.246,A -85,B 0,C 180,E1 11546.425,E2 11546.425} C_VEL
LIN {X 0,Y 266.985,Z 956.179,A -85,B 0,C 180,E1 11541.748,E2 11541.748} C_VEL
LIN {X 0,Y 274.537,Z 944.375,A -85,B 0,C 180,E1 11537.377,E2 11537.377} C_VEL
LIN {X 0,Y 283.134,Z 931.117,A -85,B 0,C 180,E1 11533.375,E2 11533.375} C_VEL
LIN {X 0,Y 291.846,Z 917.214,A -85,B 0,C 180,E1 11529.964,E2 11529.964} C_VEL
LIN {X 0,Y 301.975,Z 900.396,A -85,B 0,C 180,E1 11526.601,E2 11526.601} C_VEL
LIN {X 0,Y 311.666,Z 883.383,A -85,B 0,C 180,E1 11523.827,E2 11523.827} C_VEL
LIN {X 0,Y 320.74,Z 865.925,A -85,B 0,C 180,E1 11521.51,E2 11521.51} C_VEL
LIN {X 0,Y 329.653,Z 847.535,A -85,B 0,C 180,E1 11519.479,E2 11519.479} C_VEL
LIN {X 0,Y 338.242,Z 827.475,A -85,B 0,C 180,E1 11517.685,E2 11517.685} C_VEL
LIN {X 0,Y 346.06,Z 806.942,A -85,B 0,C 180,E1 11516.19,E2 11516.19} C_VEL
LIN {X 0,Y 352.457,Z 787.514,A -85,B 0,C 180,E1 11515.045,E2 11515.045} C_VEL
LIN {X 0,Y 358.704,Z 764.961,A -85,B 0,C 180,E1 11513.989,E2 11513.989} C_VEL
LIN {X 0,Y 363.16,Z 745.058,A -85,B 0,C 180,E1 11513.264,E2 11513.264} C_VEL
LIN {X 0,Y 367.309,Z 720.416,A -85,B 0,C 180,E1 11512.601,E2 11512.601} C_VEL
LIN {X 0,Y 387.847,Z 544.509,A -85,B 0,C 180,E1 11508.965,E2 11508.965} C_VEL
LIN {X 0,Y 386.936,Z 541.862,A -85,B 0,C 180,E1 11507.464,E2 11507.464} C_VEL
LIN {X 0,Y 386.266,Z 538.532,A -85,B 0,C 180,E1 11504.229,E2 11504.229} C_VEL
LIN {X 0,Y 386.27,Z 539.922,A -85,B 0,C 180,E1 11502.838,E2 11502.838} C_VEL
LIN {X 0,Y 387.186,Z 542.626,A -85,B 0,C 180,E1 11500.493,E2 11500.493} C_VEL
LIN {X 0,Y 387.868,Z 544.836,A -85,B 0,C 180,E1 11499.415,E2 11499.415} C_VEL
LIN {X 0,Y 366.127,Z 731.282,A -85,B 0,C 180,E1 11495.545,E2 11495.545} C_VEL
LIN {X 0,Y 361.726,Z 755.211,A -85,B 0,C 180,E1 11494.91,E2 11494.91} C_VEL
LIN {X 0,Y 355.793,Z 779.522,A -85,B 0,C 180,E1 11494.068,E2 11494.068} C_VEL
LIN {X 0,Y 349.37,Z 801.204,A -85,B 0,C 180,E1 11493.065,E2 11493.065} C_VEL
LIN {X 0,Y 341.636,Z 823.145,A -85,B 0,C 180,E1 11491.76,E2 11491.76} C_VEL
LIN {X 0,Y 333.486,Z 843.787,A -85,B 0,C 180,E1 11490.23,E2 11490.23} C_VEL
LIN {X 0,Y 323.939,Z 864.987,A -85,B 0,C 180,E1 11488.255,E2 11488.255} C_VEL
LIN {X 0,Y 313.627,Z 885.893,A -85,B 0,C 180,E1 11485.828,E2 11485.828} C_VEL
